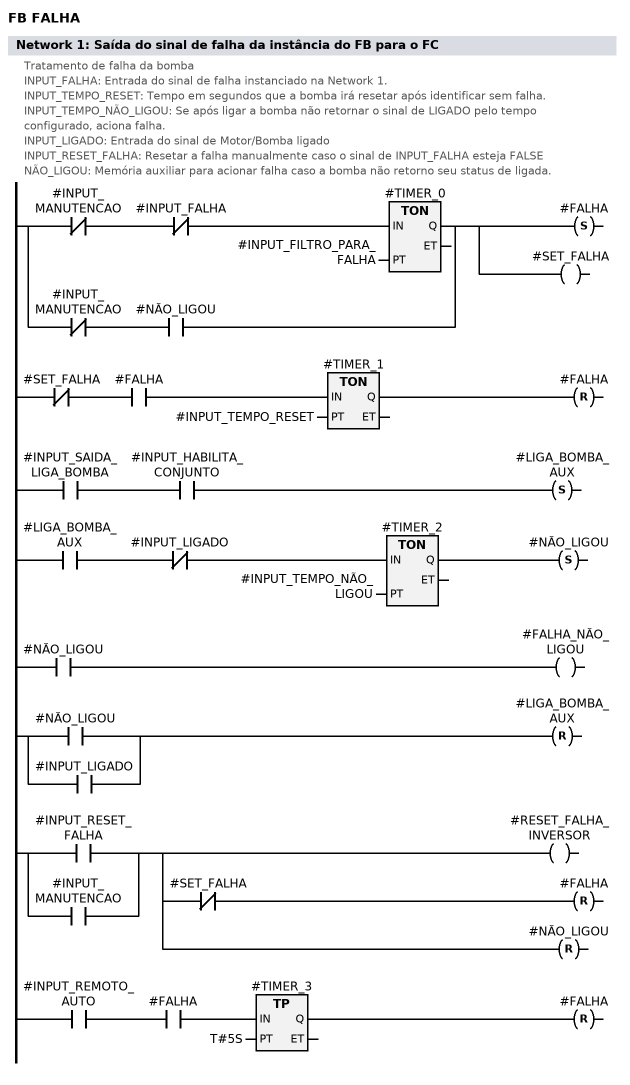
   #TIMER_0.TON(IN := NOT #INPUT_MANUTENCAO AND NOT #INPUT_FALHA, PT := #INPUT_FILTRO_PARA_FALHA);
   #_w1 := #TIMER_0.Q OR (NOT #INPUT_MANUTENCAO AND #NÃO_LIGOU);
   IF #_w1 THEN #FALHA := TRUE; END_IF;
   #SET_FALHA := #_w1;
   #TIMER_1.TON(IN := NOT #SET_FALHA AND #FALHA, PT := #INPUT_TEMPO_RESET);
   IF #TIMER_1.Q THEN #FALHA := FALSE; END_IF;
   IF #INPUT_SAIDA_LIGA_BOMBA AND #INPUT_HABILITA_CONJUNTO THEN #LIGA_BOMBA_AUX := TRUE; END_IF;
   #TIMER_2.TON(IN := #LIGA_BOMBA_AUX AND NOT #INPUT_LIGADO, PT := #INPUT_TEMPO_NÃO_LIGOU);
   IF #TIMER_2.Q THEN #NÃO_LIGOU := TRUE; END_IF;
   #FALHA_NÃO_LIGOU := #NÃO_LIGOU;
   IF #NÃO_LIGOU OR #INPUT_LIGADO THEN #LIGA_BOMBA_AUX := FALSE; END_IF;
   #RESET_FALHA_INVERSOR := #INPUT_RESET_FALHA OR #INPUT_MANUTENCAO;
   IF #RESET_FALHA_INVERSOR AND NOT #SET_FALHA THEN #FALHA := FALSE; END_IF;
   IF #RESET_FALHA_INVERSOR THEN #NÃO_LIGOU := FALSE; END_IF;
   #TIMER_3.TP(IN := #INPUT_REMOTO_AUTO AND #FALHA, PT := T#5S);
   IF #TIMER_3.Q THEN #FALHA := FALSE; END_IF;
END_REGION
END_FUNCTION_BLOCK

// folder: 1. FB Bilbiotecas/1.5 Diagnóstico

FUNCTION_BLOCK "PROFINET_DEVICE_STATES"   // FB21, SCL
{ S7_Optimized_Access := 'TRUE' }
VERSION : 0.1
   VAR_INPUT
      "Array" : Array[0..1023] of Bool;   // Array DeviceStates (1023 bools)
   END_VAR
   VAR_OUTPUT
      Word_1 : Word;   // Word 1 de saída para obter as desconecções Profinet
      Word_2 : Word;   // Word 2 de saída para obter as desconecções Profinet
   END_VAR
BEGIN
   // Word Alarmes de Desconexão Profinet

   // Word 1
   #"Word_1".%X4 := NOT #Array[4];
   #"Word_1".%X5 := NOT #Array[5];
   #"Word_1".%X6 := NOT #Array[6];
   #"Word_1".%X7 := NOT #Array[7];
   #"Word_1".%X8 := NOT #Array[8];
   #"Word_1".%X9 := NOT #Array[9];
   #"Word_1".%X10 := NOT #Array[10];
   #"Word_1".%X11 := NOT #Array[11];
   #"Word_1".%X12 := NOT #Array[12];
   #"Word_1".%X13 := NOT #Array[13];
   #"Word_1".%X14 := NOT #Array[14];
   #"Word_1".%X15 := NOT #Array[15];

   // Word 2
   #"Word_2".%X0 := NOT #Array[16];
   #"Word_2".%X1 := NOT #Array[17];
   #"Word_2".%X2 := NOT #Array[18];
   #"Word_2".%X3 := NOT #Array[19];
END_FUNCTION_BLOCK

FUNCTION_BLOCK "FB PROFINET DEVICE STATES to Word"   // FB23, SCL
{ S7_Optimized_Access := 'TRUE' }
VERSION : 0.1
   VAR_INPUT
      "Array" : Array[0..1023] of Bool;   // Array DeviceStates (1023 bools)
   END_VAR
   VAR_OUTPUT
      WORD_1 : Word;   // Word 1 de saída para obter as desconecções Profinet
      WORD_2 : Word;   // Word 2 de saída para obter as desconecções Profinet
      WORD_3 : Word;   // Word 3 de saída para obter as desconecções Profinet
      WORD_4 : Word;   // Word 4 de saída para obter as desconecções Profinet
   END_VAR
   VAR
      "word" : Array[1..4] of Word;
      i : Int;
      j : Int;
   END_VAR
BEGIN
   // Word Alarmes de Desconexão Profinet




   // Word 1
   #WORD_1.%X0 := NOT #Array[0];
   #WORD_1.%X1 := NOT #Array[1];
   #WORD_1.%X2 := NOT #Array[2];
   #WORD_1.%X3 := NOT #Array[3];
   #WORD_1.%X4 := NOT #Array[4];(*
   #WORD_1.%X5 := NOT #Array[5];
   #WORD_1.%X6 := NOT #Array[6];
   #WORD_1.%X7 := NOT #Array[7];
   #WORD_1.%X8 := NOT #Array[8];
   #WORD_1.%X9 := NOT #Array[9];*)
   #WORD_1.%X10 := NOT #Array[10];
   #WORD_1.%X11 := NOT #Array[11];
   #WORD_1.%X12 := NOT #Array[12];
   #WORD_1.%X13 := NOT #Array[13];(*
   #WORD_1.%X14 := NOT #Array[14];
   #WORD_1.%X15 := NOT #Array[15];

   //Word 2
   #WORD_2.%X0 := NOT #Array[16];
   #WORD_2.%X1 := NOT #Array[17];
   #WORD_2.%X2 := NOT #Array[18];
   #WORD_2.%X3 := NOT #Array[19];*)
   #WORD_2.%X4 := NOT #Array[20];
   #WORD_2.%X5 := NOT #Array[21];
   #WORD_2.%X6 := NOT #Array[22];
   #WORD_2.%X7 := NOT #Array[23];
   #WORD_2.%X8 := NOT #Array[24];
   #WORD_2.%X9 := NOT #Array[25];
   #WORD_2.%X10 := NOT #Array[26];
   #WORD_2.%X11 := NOT #Array[27];
   #WORD_2.%X12 := NOT #Array[28];
   #WORD_2.%X13 := NOT #Array[29];
   #WORD_2.%X14 := NOT #Array[30];
   #WORD_2.%X15 := NOT #Array[31];

   //Word 3
   #WORD_3.%X0 := NOT #Array[32];
   #WORD_3.%X1 := NOT #Array[33];
   #WORD_3.%X2 := NOT #Array[34];
   #WORD_3.%X3 := NOT #Array[35];(*
   #WORD_3.%X4 := NOT #Array[36];
   #WORD_3.%X5 := NOT #Array[37];
   #WORD_3.%X6 := NOT #Array[38];
   #WORD_3.%X7 := NOT #Array[39];*)
   #WORD_3.%X8 := NOT #Array[40];
   #WORD_3.%X9 := NOT #Array[41];
   #WORD_3.%X10 := NOT #Array[42];
   #WORD_3.%X11 := NOT #Array[43];
   #WORD_3.%X12 := NOT #Array[44];
   #WORD_3.%X13 := NOT #Array[45];
   #WORD_3.%X14 := NOT #Array[46];
   #WORD_3.%X15 := NOT #Array[47];

   //Word 4
   #WORD_4.%X0 := NOT #Array[48];(*
   #WORD_4.%X1 := NOT #Array[49];*)
   #WORD_4.%X2 := NOT #Array[50];
   #WORD_4.%X3 := NOT #Array[51];
   #WORD_4.%X4 := NOT #Array[52];
   #WORD_4.%X5 := NOT #Array[53];
   #WORD_4.%X6 := NOT #Array[54];
   #WORD_4.%X7 := NOT #Array[55];
   #WORD_4.%X8 := NOT #Array[56];
   #WORD_4.%X9 := NOT #Array[57];
   #WORD_4.%X10 := NOT #Array[58];
   #WORD_4.%X11 := NOT #Array[59];
   #WORD_4.%X12 := NOT #Array[60];
   #WORD_4.%X13 := NOT #Array[61];(*
   #WORD_4.%X14 := NOT #Array[62];
   #WORD_4.%X15 := NOT #Array[63];*)
END_FUNCTION_BLOCK

FUNCTION_BLOCK "FB PROFINET DEVICE STATES to BIT"   // FB26, SCL
{ S7_Optimized_Access := 'TRUE' }
VERSION : 0.1
   VAR_INPUT
      "Array" : Array[0..1023] of Bool;   // Array DeviceStates (1023 bools)
   END_VAR
   VAR_OUTPUT
      Bit_1 : Bool;   // Word 1 de saída para obter as desconecções Profinet
      Bit_2 : Bool;   // Word 2 de saída para obter as desconecções Profinet
      Bit_3 : Bool;   // Word 3 de saída para obter as desconecções Profinet
      Bit_4 : Bool;   // Word 4 de saída para obter as desconecções Profinet
      Bit_5 : Bool;
      Bit_6 : Bool;
      Bit_7 : Bool;
      Bit_8 : Bool;
      Bit_9 : Bool;
      Bit_10 : Bool;
      Bit_11 : Bool;
      Bit_12 : Bool;
      Bit_13 : Bool;
      Bit_14 : Bool;
      Bit_15 : Bool;
      Bit_16 : Bool;
      Bit_17 : Bool;
      Bit_18 : Bool;
      Bit_19 : Bool;
      Bit_20 : Bool;
      Bit_21 : Bool;
      Bit_22 : Bool;
      Bit_23 : Bool;
      Bit_24 : Bool;
      Bit_25 : Bool;
      Bit_26 : Bool;
      Bit_27 : Bool;
      Bit_28 : Bool;
      Bit_29 : Bool;
      Bit_30 : Bool;
      Bit_31 : Bool;
      Bit_32 : Bool;
      Bit_33 : Bool;
      Bit_34 : Bool;
      Bit_35 : Bool;
      Bit_36 : Bool;
      Bit_37 : Bool;
      Bit_38 : Bool;
      Bit_39 : Bool;
      Bit_40 : Bool;
      Bit_41 : Bool;
      Bit_42 : Bool;
      Bit_43 : Bool;
      Bit_44 : Bool;
      Bit_45 : Bool;
      Bit_46 : Bool;
      Bit_47 : Bool;
      Bit_48 : Bool;
      Bit_49 : Bool;
      Bit_50 : Bool;
      Bit_51 : Bool;
      Bit_52 : Bool;
      Bit_53 : Bool;
      Bit_54 : Bool;
      Bit_55 : Bool;
      Bit_56 : Bool;
      Bit_57 : Bool;
      Bit_58 : Bool;
      Bit_59 : Bool;
      Bit_60 : Bool;
      Bit_61 : Bool;
      Bit_62 : Bool;
      Bit_63 : Bool;
      Bit_64 : Bool;
   END_VAR
   VAR
      "word" : Array[1..4] of Word;
      i : Int;
      j : Int;
   END_VAR
BEGIN
   #Bit_1 :=  #Array[0];
   #Bit_2 :=  #Array[1];
   #Bit_3 :=  #Array[2];
   #Bit_4 :=  #Array[3];
   #Bit_5 :=  #Array[4];
   #Bit_6 :=  #Array[5];
   #Bit_7 :=  #Array[6];
   #Bit_8 :=  #Array[7];
   #Bit_9 :=  #Array[8];
   #Bit_10 :=  #Array[9];
   #Bit_11 :=  #Array[10];
   #Bit_12 :=  #Array[11];
   #Bit_13 :=  #Array[12];
   #Bit_14 :=  #Array[13];
   #Bit_15 :=  #Array[14];
   #Bit_16 :=  #Array[15];
   #Bit_17 :=  #Array[16];
   #Bit_18 :=  #Array[17];
   #Bit_19 :=  #Array[18];
   #Bit_20 :=  #Array[19];
   #Bit_21 :=  #Array[20];
   #Bit_22 :=  #Array[21];
   #Bit_23 :=  #Array[22];
   #Bit_24 :=  #Array[23];
   #Bit_25 :=  #Array[24];
   #Bit_26 :=  #Array[25];
   #Bit_27 :=  #Array[26];
   #Bit_28 :=  #Array[27];
   #Bit_29 :=  #Array[28];
   #Bit_30 :=  #Array[29];
   #Bit_31 :=  #Array[30];
   #Bit_32 :=  #Array[31];
   #Bit_33 :=  #Array[32];
   #Bit_34 :=  #Array[33];
   #Bit_35 :=  #Array[34];
   #Bit_36 :=  #Array[35];
   #Bit_37 :=  #Array[36];
   #Bit_38 :=  #Array[37];
   #Bit_39 :=  #Array[38];
   #Bit_40 :=  #Array[39];
   #Bit_41 :=  #Array[40];
   #Bit_42 :=  #Array[41];
   #Bit_43 :=  #Array[42];
   #Bit_44 :=  #Array[43];
   #Bit_45 :=  #Array[44];
   #Bit_46 :=  #Array[45];
   #Bit_47 :=  #Array[46];
   #Bit_48 :=  #Array[47];
   #Bit_49 :=  #Array[48];
   #Bit_50 :=  #Array[49];
   #Bit_51 :=  #Array[50];
   #Bit_52 :=  #Array[51];
   #Bit_53 :=  #Array[52];
   #Bit_54 :=  #Array[53];
   #Bit_55 :=  #Array[54];
   #Bit_56 :=  #Array[55];
   #Bit_57 :=  #Array[56];
   #Bit_58 :=  #Array[57];
   #Bit_59 :=  #Array[58];
   #Bit_60 :=  #Array[59];
   #Bit_61 :=  #Array[60];
   #Bit_62 :=  #Array[61];
   #Bit_63 :=  #Array[62];
   #Bit_64 :=  #Array[63];
END_FUNCTION_BLOCK

FUNCTION_BLOCK "FB DIAG MODULES"   // FB28, LAD
{ S7_Optimized_Access := 'TRUE' }
VERSION : 0.1
   VAR_INPUT
      LADDR : HW_ANY;   // ID de hardware do componente de hardware
      MODE : UInt;   // Use o parâmetro de modo para selecionar quais dados de diagnóstico são emitidos.
   END_VAR
   VAR_OUTPUT
      "OUT_WORD[bit]" : Bool;   // Bit da Word de saída representando falha/avaria do dispositivo
      Maintence_State : String;
      Component_StateDetail : String;
      Own_State : String;
      IO_State : String;
      Operating_State : String;
      Ret_Val : String;
   END_VAR
   VAR
      "Maintence State" : Array[0..10] of String;
      ComponentStateDetail : Array[0..31] of String;
      OwnState : Array[0..7] of String;
      IOState : Array[0..15] of String;
      OperatingState : Array[0..40] of String;
      DIAG : DIS;
      CNT_DIAG : UInt;
      RET_VAL_STRING : Array[0..6] of String;
      RET_VAL_1 : Int;
   END_VAR
   // "Maintence State"[0] := 'Good';
   // "Maintence State"[1] := 'The hardware component is disabled.';
   // "Maintence State"[5] := 'Maintenance required';
   // "Maintence State"[6] := 'Maintenance demanded';
   // "Maintence State"[7] := 'Error';
   // "Maintence State"[8] := 'Status unknown / error in higher-level hardware component';
   // "Maintence State"[10] := 'Inputs/outputs are not available.';
   // ComponentStateDetail[3] := 'least one qualified diagnostics is available';
   // ComponentStateDetail[4] := 'Maintenance required for at least one channel or the component';
   // ComponentStateDetail[5] := 'Maintenance demanded for at least one channel or the component';
   // ComponentStateDetail[6] := 'Error in at least one channel or the component';
   // ComponentStateDetail[7] := 'Application Ready Pending - No I/O access';
   // ComponentStateDetail[8] := 'Locked by Superordinated - No access to hardware component';
   // ComponentStateDetail[9] := 'Locked by IOController - No access to hardware component';
   // ComponentStateDetail[10] := 'Locked by IOSupervisor - No access to hardware component';
   // ComponentStateDetail[16] := 'Submodule or module disabled';
   // ComponentStateDetail[17] := 'CiR operation active';
   // ComponentStateDetail[18] := 'Input not available';
   // ComponentStateDetail[19] := 'Output not available';
   // ComponentStateDetail[20] := 'Overflow diagnostics buffer';
   // ComponentStateDetail[21] := 'Diagnostics not available';
   // ComponentStateDetail[22] := 'Partial device failure (with PNIO for Shared iDevices)';
   // OwnState[0] := 'Good';
   // OwnState[1] := 'Disabled';
   // OwnState[2] := 'Maintenance required';
   // OwnState[3] := 'Maintenance demanded';
   // OwnState[4] := 'Error';
   // OwnState[5] := 'Not accessible';
   // OwnState[6] := 'Diagnostic status unknown';
   // OwnState[7] := 'IO not available - Inputs/outputs are not available.';
   // IOState[0] := 'Good';
   // IOState[1] := 'Disabled';
   // IOState[2] := 'Maintenance required';
   // IOState[3] := 'Maintenance demanded';
   // IOState[4] := 'Error';
   // IOState[5] := 'Hardware component not reachable - Hardware component cannot be accessed.';
   // IOState[6] := 'Qualified: Bit 6 = 1 if at least one qualified diagnostics is available';
   // IOState[7] := 'I/O data not available - I/O data not available';
   // IOState[14] := 'Network error';
   // IOState[15] := 'Hardware error';
   // OperatingState[1] := 'STOP / firmware update';
   // OperatingState[2] := 'STOP / Memory reset';
   // OperatingState[3] := 'STOP / self start';
   // OperatingState[4] := 'STOP';
   // OperatingState[5] := 'Memory reset';
   // OperatingState[6] := 'Startup';
   // OperatingState[8] := 'RUN';
   // OperatingState[9] := 'RUN-Redundant';
   // OperatingState[10] := 'HOLD';
   // OperatingState[13] := 'DEFECT (Note: can only be seen in diagnostics buffer entries)';
   // OperatingState[15] := 'De-energized (Note: can only be seen in diagnostics buffer entries)';
   // OperatingState[16] := 'CiR';
   // OperatingState[17] := 'STOP without ODIS';
   // OperatingState[18] := 'RUN ODIS';
   // OperatingState[19] := 'PgmTest';
   // OperatingState[20] := 'RunPgmTest (state of primary CPU when the backup CPU is in test mode)';
   // OperatingState[21] := 'Run-Syncup (only Primary CPU in SYNCUP system state)';
   // OperatingState[22] := 'SYNCUP (only backup CPU in SYNCUP system state)';
   // OperatingState[31] := 'State of partner CPU unknown (for example when the partner CPU is not available)';
   // OperatingState[33] := 'STOP system state';
   // OperatingState[35] := 'STARTUP system state';
   // OperatingState[37] := 'RUN-Solo system state';
   // OperatingState[38] := 'SYNCUP system state';
   // OperatingState[40] := 'RUN-Redundant system state';
   // RET_VAL_STRING[0] := 'Feedback signal ok';
   // RET_VAL_STRING[1] := 'The data area at the DETAIL parameter is too small. Not all details of the diagnostics data are output.';
   // RET_VAL_STRING[2] := 'Value in the MODE parameter is not supported.';
   // RET_VAL_STRING[3] := 'Type at the DIAG parameter is not supported with the selected mode (parameter MODE).';
   // RET_VAL_STRING[4] := 'Type at the DETAIL parameter is not supported with the selected mode (parameter MODE).';
   // RET_VAL_STRING[5] := 'LADDR does not exist';
   // RET_VAL_STRING[6] := 'Insufficient resources for parallel execution.';
BEGIN

REGION Network 1
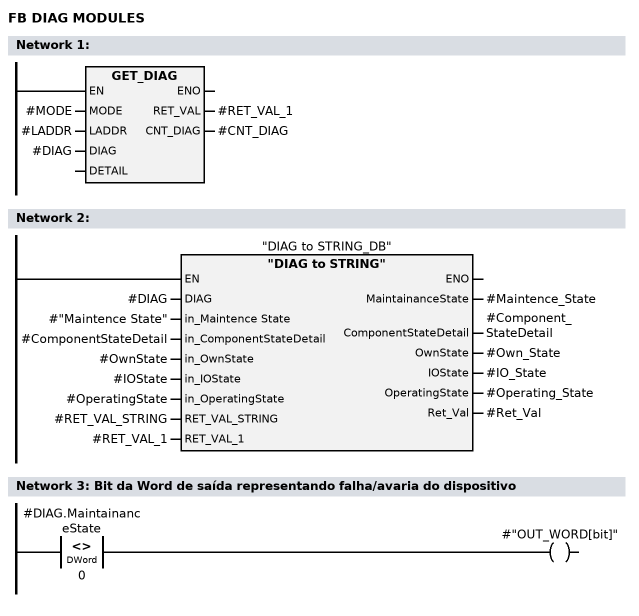
   #RET_VAL_1 := GET_DIAG(MODE := #MODE, LADDR := #LADDR, DIAG := #DIAG, CNT_DIAG => #CNT_DIAG);
END_REGION

REGION Network 2
   RUNG wire#powerrail
      "DIAG to STRING_DB"(DIAG := #DIAG, "in_Maintence State" := #"Maintence State", in_ComponentStateDetail := #ComponentStateDetail, in_OwnState := #OwnState, in_IOState := #IOState, in_OperatingState := #OperatingState, RET_VAL_STRING := #RET_VAL_STRING, RET_VAL_1 := #RET_VAL_1, MaintainanceState => #Maintence_State, ComponentStateDetail => #Component_StateDetail, OwnState => #Own_State, IOState => #IO_State, OperatingState => #Operating_State, Ret_Val => #Ret_Val)
   END_RUNG
   // the same network as SCL:
   "DIAG to STRING_DB"(DIAG := #DIAG,   // "DIAG to STRING"
                       "in_Maintence State" := #"Maintence State",
                       in_ComponentStateDetail := #ComponentStateDetail,
                       in_OwnState := #OwnState,
                       in_IOState := #IOState,
                       in_OperatingState := #OperatingState,
                       RET_VAL_STRING := #RET_VAL_STRING,
                       RET_VAL_1 := #RET_VAL_1,
                       MaintainanceState => #Maintence_State,
                       ComponentStateDetail => #Component_StateDetail,
                       OwnState => #Own_State,
                       IOState => #IO_State,
                       OperatingState => #Operating_State,
                       Ret_Val => #Ret_Val);
END_REGION

REGION Network 3: Bit da Word de saída representando falha/avaria do dispositivo
   RUNG wire#powerrail
      { S7_Templates := "SrcType := DWord" } NE_Contact(in1 := #DIAG.MaintainanceState, in2 := 0)
      Coil( #"OUT_WORD[bit]" )
   END_RUNG
   // the same network as SCL:
   #"OUT_WORD[bit]" := #DIAG.MaintainanceState <> 0;
END_REGION
END_FUNCTION_BLOCK

FUNCTION_BLOCK "DIAG to STRING"   // FB29, SCL
{ S7_Optimized_Access := 'TRUE' }
VERSION : 0.1
   VAR_INPUT
      DIAG : DIS;
      "in_Maintence State" : Array[0..10] of String;
      in_ComponentStateDetail : Array[0..31] of String;
      in_OwnState : Array[0..7] of String;
      in_IOState : Array[0..15] of String;
      in_OperatingState : Array[0..40] of String;
      RET_VAL_STRING : Array[0..6] of String;
      RET_VAL_1 : UInt;
   END_VAR
   VAR_OUTPUT
      MaintainanceState : String[254];
      ComponentStateDetail : String[254];
      OwnState : String[254];
      IOState : String[254];
      OperatingState : String[254];
      Ret_Val : String[254];
   END_VAR
   VAR
      i : Int;
      j : UInt;
      k : UInt;
      "m" : UInt;
      n : UInt;
      o : UInt;
      Separator : String[5];
   END_VAR
BEGIN
   // PARA MaintainanceState
   FOR #i := 0 TO 10 DO
       IF #DIAG.MaintainanceState = #i THEN
           #MaintainanceState := #"in_Maintence State"[#i];
       END_IF;
   END_FOR;

   #Separator := '; ';
   #ComponentStateDetail := '';
   #IOState := '';
   FOR #j := 0 TO 31 DO
       // testa se o bit #j está 1
       IF (#DIAG.ComponentStateDetail AND SHL(IN:= DWORD#1, N:= #j)) <> DWORD#0 THEN
           // ignora entradas vazias
           IF LEN(#in_ComponentStateDetail[#j]) > 0 THEN
               // separador só se já houver conteúdo
               IF LEN(#ComponentStateDetail) > 0 THEN
                   #ComponentStateDetail := CONCAT(IN1 := #ComponentStateDetail, IN2 := #Separator);
               END_IF;
               // concatena o texto do índice ativo
               #ComponentStateDetail := CONCAT(IN1 := #ComponentStateDetail, IN2 := #in_ComponentStateDetail[#j]);
           END_IF;
       END_IF;
   END_FOR;

   FOR #k := 0 TO 7 DO
       IF #DIAG.OwnState = #k THEN
           #OwnState := #in_OwnState[#k];
       END_IF;
   END_FOR;

   FOR #m := 0 TO 15 DO
       IF (#DIAG.IOState AND SHL(IN := DWORD#1, N := #m)) <> DWORD#0 THEN
           IF LEN(#in_IOState[#m]) > 0 THEN
               IF LEN(#IOState) > 0 THEN
                   #IOState := CONCAT(IN1 := #IOState, IN2 := #Separator);
               END_IF;
               #IOState := CONCAT(IN1 := #IOState, IN2 := #in_IOState[#m]);
           END_IF;
       END_IF;
   END_FOR;

   FOR #n := 0 TO 40 DO
       IF #DIAG.OperatingState = #n THEN
           #OperatingState := #in_OperatingState[#i];
       END_IF;
   END_FOR;

   CASE #RET_VAL_1 OF
       UINT#16#0000:
           #Ret_Val := #RET_VAL_STRING[0];
       UINT#16#8080:
           #Ret_Val := #RET_VAL_STRING[2];
       UINT#16#8081:
           #Ret_Val := #RET_VAL_STRING[3];
       UINT#16#8082:
           #Ret_Val := #RET_VAL_STRING[4];
       UINT#16#8090:
           #Ret_Val := #RET_VAL_STRING[5];
       UINT#16#80C1:
           #Ret_Val := #RET_VAL_STRING[6];

       ELSE
           #Ret_Val := #RET_VAL_STRING[2];  // default
   END_CASE;
END_FUNCTION_BLOCK

// folder: 1. FB Bilbiotecas/1.6 Comunicação Modbus

FUNCTION_BLOCK "FB MODBUS MASTER BLOCK MMW"   // FB18, LAD
{ S7_Optimized_Access := 'TRUE' }
VERSION : 0.1
// Instanciamento do Bloco Modbus Master para cada Driver (Multimedidor)
// 
// Network 1: Chamada por índice de endereço
// Network 2: Falha de comunicação Modbus
// Network 3: Reset do módulo de comunicação Modbus
   VAR_INPUT
      INDEX_DRIVER : Int;   // Índice do driver, numerando a instância de cada um
      INDEX_ADDR : Int;   // Índice do endereço, numerando a ordem de leitura de cada um
      TRIGGER : Bool;   // Gatilho de chamada do bloco. (Recebido da instância do FB SCAN DRIVERS conforme o DONE do bloco master)
      MODBUS_ID : Int;   // Endereço ID do Modbus
      ARRAY_ADDR_MMW : Array[0..38] of Int;   // Array de endereços (Todos os 41 endereços cadastrados na tabela Modbus do equipamento)
      INDEX_BLOCK : Int;   // Índice de instância, para definir quando os blocos Master serão chamados
      CICLE_TIMES_SET_ALARME : Int;   // Cadastro do "Tryout", número de tentativas de comunicação antes de acionar o erro
   END_VAR
   VAR_OUTPUT
      DRIVER_ERROR_COMUNIC : Bool;   // Erro de comunicação Modbus
      ERROR_CODE : Word;   // Código do erro de comunicação Modbus
      RESET_PTP : Bool;   // Saída para reset do módulo Commload
   END_VAR
   VAR_IN_OUT
      MODBUS_MASTER : Modbus_Master;
      ARRAY_MMW : Array[0..38] of Real;   // Array da DB GLOBAL onde os registros são armazenados
   END_VAR
   VAR
      PULSE_SCAN : Bool;   // Pulso para contagem do número de tentativas de comunicação mal sucedidas
      COUT_PULSE : Bool;   // Memória auxiliar do pulso
      ERROR_CICLES : Int;   // Memória de incremento a cada pulso do PULSE_SCAN
      ACTUAL_ERROR : Word;   // Captura do código de erro na tentativa de comunicação mal sucedida
      MASTER_DRIVER_LAST_ERROR : Int;   // Índice do driver que registrou o último erro
      ARRAY_READ_MMW : Array[0..254] of Real;   // Array local para armazenar temporariamente as leituras antes de mover à DB GLOBAL
      HABILITA_RESET : Bool;   // Habilita reset após intervalo de tempo
      AUX_RESET : Bool;   // Memória auxiliar para o reset modbus
      RESET_TIMER_1 : IEC_TIMER;   // Tempo de cooldown para utilizar o reset novamente
      RESET_TIMER_2 : IEC_TIMER;   // Tempo de saída acionada (reset)
   END_VAR
   VAR_TEMP   // added for the SCL form of the ladder/FBD networks
      _w1 : Bool;
      _w2 : Bool;
   END_VAR
BEGIN

REGION Network 1: Function BLock MODBUS MASTER BLOCK MMW
   // Ao chamar o bloco, o índice de endereço irá alternar entre os 41 endereços do multimedidor. Essas informações são registradas em um array de tamanho 41 e movidos à DB GLOBAL.
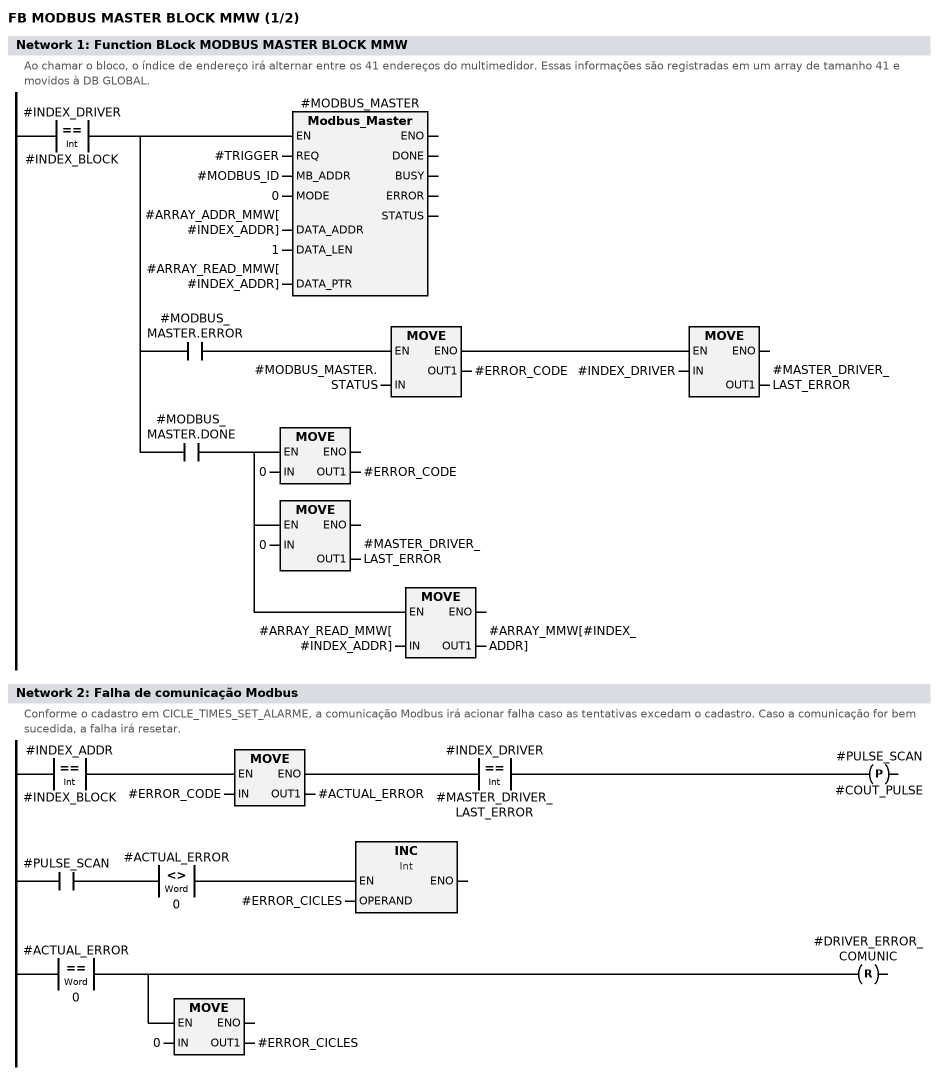
   #_w1 := #INDEX_DRIVER = #INDEX_BLOCK;
   IF #_w1 THEN
       #MODBUS_MASTER(REQ := #TRIGGER,   // Modbus_Master
                      MB_ADDR := #MODBUS_ID,
                      MODE := 0,
                      DATA_ADDR := #ARRAY_ADDR_MMW[#INDEX_ADDR],
                      DATA_LEN := 1,
                      DATA_PTR := #ARRAY_READ_MMW[#INDEX_ADDR]);
   END_IF;
   IF #_w1 AND #MODBUS_MASTER.ERROR THEN
       #ERROR_CODE := #MODBUS_MASTER.STATUS;
       #MASTER_DRIVER_LAST_ERROR := #INDEX_DRIVER;
   END_IF;
   IF #_w1 AND #MODBUS_MASTER.DONE THEN
       #ERROR_CODE := 0;
       #MASTER_DRIVER_LAST_ERROR := 0;
       #ARRAY_MMW[#INDEX_ADDR] := #ARRAY_READ_MMW[#INDEX_ADDR];
   END_IF;
END_REGION

REGION Network 2: Falha de comunicação Modbus
   // Conforme o cadastro em CICLE_TIMES_SET_ALARME, a comunicação Modbus irá acionar falha caso as tentativas excedam o cadastro. Caso a comunicação for bem sucedida, a falha irá resetar.
   #_w1 := #INDEX_ADDR = #INDEX_BLOCK;
   IF #_w1 THEN #ACTUAL_ERROR := #ERROR_CODE; END_IF;
   #_w2 := #_w1 AND (#INDEX_DRIVER = #MASTER_DRIVER_LAST_ERROR);
   #PULSE_SCAN := #_w2 AND NOT #COUT_PULSE;   // rising edge
   #COUT_PULSE := #_w2;
   IF #PULSE_SCAN AND (#ACTUAL_ERROR <> 0) THEN #ERROR_CICLES := #ERROR_CICLES + 1; END_IF;
   IF #ACTUAL_ERROR = 0 THEN
       #DRIVER_ERROR_COMUNIC := FALSE;
       #ERROR_CICLES := 0;
   END_IF;
END_REGION

REGION Network 3: Reset do módulo de comunicação Modbus
   // Reset ao identificar erro de comunicação.
   // Tempo de cooldown 600s (10min): Intervalo de tempo após o reset para resetar novamente caso o equipamento ainda esteja em erro.
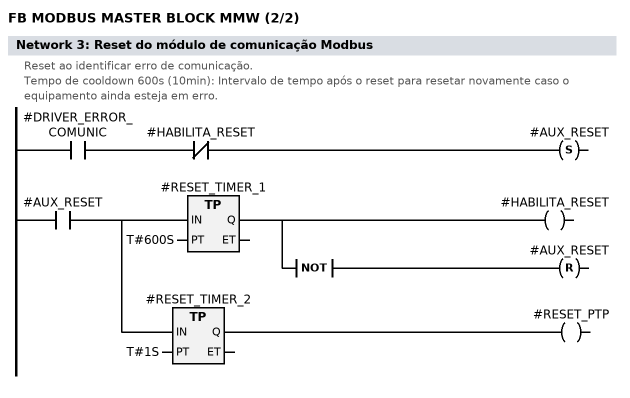
   IF #DRIVER_ERROR_COMUNIC AND NOT #HABILITA_RESET THEN #AUX_RESET := TRUE; END_IF;
   #RESET_TIMER_1.TP(IN := #AUX_RESET, PT := T#600S);
   #HABILITA_RESET := #RESET_TIMER_1.Q;
   #_w1 := #AUX_RESET;
   IF NOT #RESET_TIMER_1.Q THEN #AUX_RESET := FALSE; END_IF;
   #RESET_TIMER_2.TP(IN := #_w1, PT := T#1S);
   #RESET_PTP := #RESET_TIMER_2.Q;
END_REGION
END_FUNCTION_BLOCK

FUNCTION_BLOCK "FB MODBUS MASTER BLOCK"   // FB19, LAD
TITLE = Function Block MODBUS MASTER BLOCK
{ S7_Optimized_Access := 'TRUE' }
VERSION : 0.1
// Instanciamento do Bloco Modbus Master para cada Driver (Inversor ou rádio)
// 
// Network 1: Chamada por índice de endereço
// Network 2: Falha de comunicação Modbus
// Network 3: Segundeiro, segundos sem comunicação
// Network 4: Reset do módulo de comunicação Modbus
   VAR_INPUT
      INDEX_DRIVER : Int;   // Índice do driver, numerando a instância de cada um
      INDEX_ADDR : Int;   // Índice do endereço, numerando a ordem de leitura de cada um
      TRIGGER : Bool;   // Gatilho de chamada do bloco. (Recebido da instância do FB SCAN DRIVERS conforme o DONE do bloco master)
      MODBUS_ID : Int;   // Endereço ID do Modbus
      DATA_ADDR_1 : DInt;   // Endereço 1 para acesso à tabela modbus
      MODE_ADDR_1 : Byte;   // Modo (0 = Leitura, 1 = Escrita)
      DATA_LEN_1 : Byte;
      IS_MMW_2 : Bool;
      DATA_ADDR_2 : DInt;   // Endereço 2 para acesso à tabela modbus
      MODE_ADDR_2 : Byte;   // Modo (0 = Leitura, 1 = Escrita)
      DATA_LEN_2 : Byte;
      IS_MMW_3 : Bool;
      DATA_ADDR_3 : DInt;   // Endereço 3 para acesso à tabela modbus
      MODE_ADDR_3 : Byte;   // Modo (0 = Leitura, 1 = Escrita)
      DATA_LEN_3 : Byte;
      IS_MMW_4 : Bool;
      DATA_ADDR_4 : DInt;   // Endereço 3 para acesso à tabela modbus
      MODE_ADDR_4 : Byte;   // Modo (0 = Leitura, 1 = Escrita)
      DATA_LEN_4 : Byte;
      IS_MMW_5 : Bool;
      DATA_ADDR_5 : DInt;   // Endereço 3 para acesso à tabela modbus
      MODE_ADDR_5 : Byte;   // Modo (0 = Leitura, 1 = Escrita)
      DATA_LEN_5 : Byte;
      INDEX_BLOCK : Int;   // Índice de instância, para definir quando os blocos Master serão chamados
      CICLE_TIMES_SET_ALARME : Int;   // Cadastro do "Tryout", número de tentativas de comunicação antes de acionar o erro
   END_VAR
   VAR_OUTPUT
      DRIVER_ERROR_COMUNIC : Bool;   // Erro de comunicação Modbus
      ERROR_CODE : Word;   // Código do erro de comunicação Modbus
      ERROR_CICLES : Int;   // Memória de incremento a cada pulso do PULSE_SCAN
      SEGUNDEIRO : Int;   // Segundos sem comunicação
      RESET_PTP : Bool;   // Saída para reset do módulo Commload
   END_VAR
   VAR_IN_OUT
      MODBUS_MASTER : Modbus_Master;   // Entrada do Bloco Master na instância
      DATA_PTR_1 : Variant;   // Endereço da DB GLOBAL onde a leitura proveninente do DATA_ADDR_1 é armazenada
      DATA_PTR_2 : Variant;   // Endereço da DB GLOBAL onde a leitura proveninente do DATA_ADDR_2 é armazenada
      DATA_PTR_3 : Variant;   // Endereço da DB GLOBAL onde a leitura proveninente do DATA_ADDR_3 é armazenada
      DATA_PTR_4 : Variant;   // Endereço da DB GLOBAL onde a leitura proveninente do DATA_ADDR_3 é armazenada
      DATA_PTR_5 : Variant;   // Endereço da DB GLOBAL onde a leitura proveninente do DATA_ADDR_3 é armazenada
   END_VAR
   VAR
      PULSE_SCAN : Bool;   // Pulso para contagem do número de tentativas de comunicação mal sucedidas
      COUNT_PULSE : Bool;   // Memória auxiliar do pulso
      ACTUAL_ERROR : Word;   // Captura do código de erro na tentativa de comunicação mal sucedida
      MASTER_DRIVER_LAST_ERROR : Int;   // Índice do driver que registrou o último erro
      ERROR_MASTER_1 : Bool;   // Código de erro do mestre 1 (addr 1)
      ERROR_MASTER_2 : Bool;   // Código de erro do mestre 2 (addr 2)
      ERROR_MASTER_3 : Bool;   // Código de erro do mestre 3 (addr 3)
      ERROR_MASTER_4 : Bool;   // Código de erro do mestre 3 (addr 3)
      ERROR_MASTER_5 : Bool;   // Código de erro do mestre 3 (addr 3)
      STATUS_MASTER_1 : Word;   // Status do mestre 1 (addr 1)
      STATUS_MASTER_2 : Word;   // Status do mestre 2 (addr 2)
      STATUS_MASTER_3 : Word;   // Status do mestre 3 (addr 3)
      STATUS_MASTER_4 : Word;   // Status do mestre 3 (addr 3)
      STATUS_MASTER_5 : Word;   // Status do mestre 3 (addr 3)
      DONE : Bool;   // Indicador de comunicação bem sucedida
      DONE_PULSO : Int;   // Pulso de comunicação bem sucedida
      SEGUNDEIRO_PULSO : Bool;   // Pulso para contar os segundos sem comunicação
      SEGUNDEIRO_AUX : Bool;   // Memória auxiliar do segundeiro
      HABILITA_RESET : Bool;   // Habilita reset após intervalo de tempo
      AUX_RESET : Bool;   // Memória auxiliar para o reset modbus
      SET_COOLDOWN : Bool;   // Memória Auxiliar do Cooldown Timer
      RESET_COOLDOWN : Bool;   // Memória Auxiliar do Cooldown Timer
      RESET_TIMER_1 : IEC_TIMER;   // Tempo de cooldown para utilizar o reset novamente
      RESET_TIMER_2 : IEC_TIMER;   // Tempo de saída acionada (reset)
      COOLDOWN_TIMER_1 : IEC_TIMER;   // Tempo para resetar os ciclos sem comunicação
      COOLDOWN_TIMER_2 : IEC_TIMER;   // Tempo de espera após reset para resetar novamente
      COOLDOWN_TIMER_3 : IEC_TIMER;
   END_VAR
   VAR_TEMP   // added for the SCL form of the ladder/FBD networks
      _w1 : Bool;
      _w2 : Bool;
   END_VAR
BEGIN

REGION Network 1: Chamada por índice de endereço
   // Cada vez que o bloco Master é chamado, um índice de endereço diferente é armazenado.
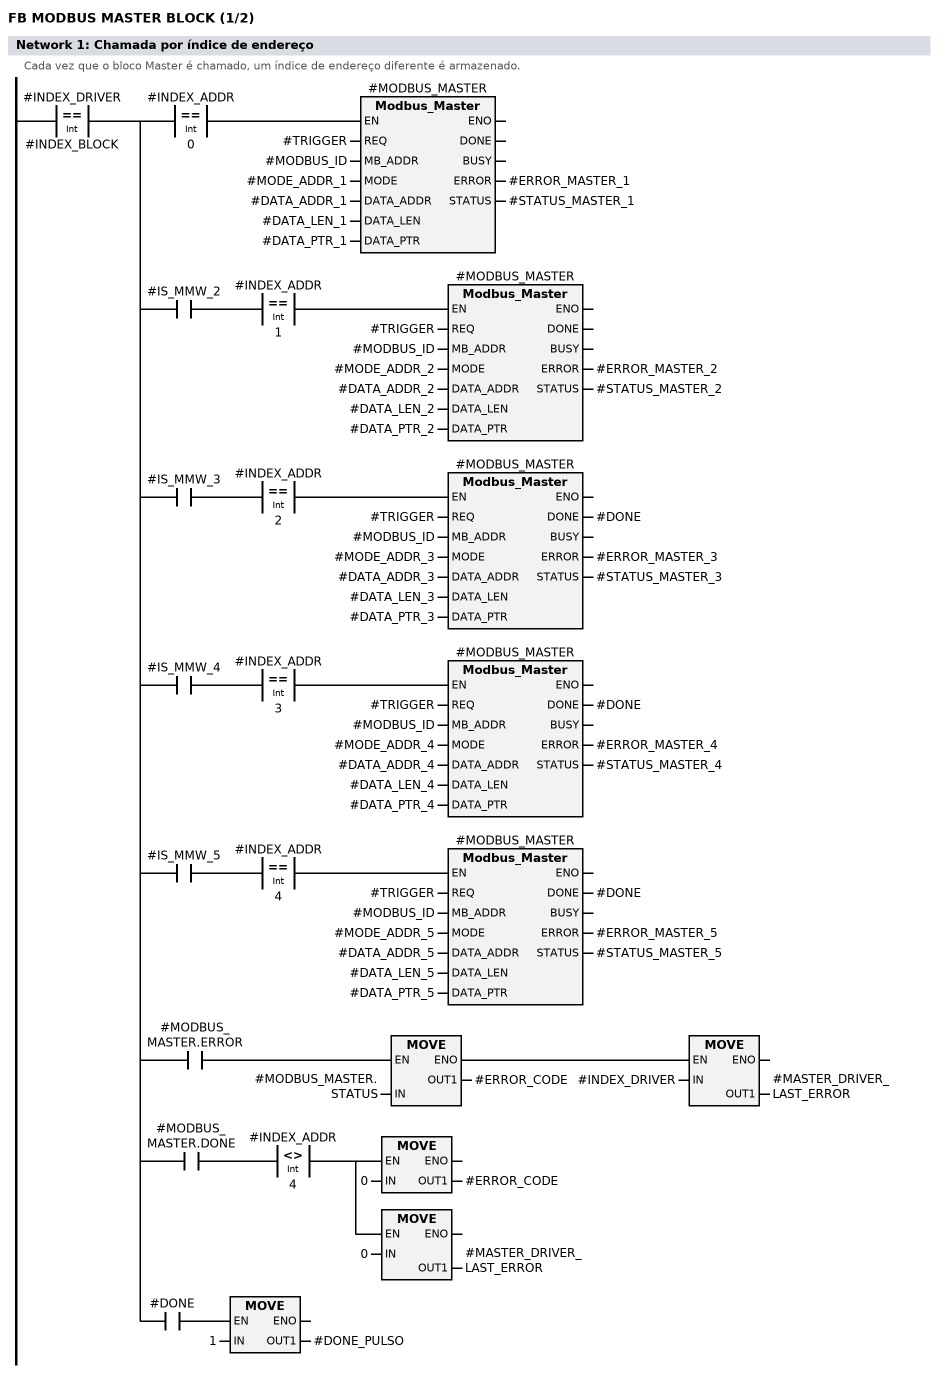
   #_w1 := #INDEX_DRIVER = #INDEX_BLOCK;
   IF #_w1 AND (#INDEX_ADDR = 0) THEN
       #MODBUS_MASTER(REQ := #TRIGGER,   // Modbus_Master
                      MB_ADDR := #MODBUS_ID,
                      MODE := #MODE_ADDR_1,
                      DATA_ADDR := #DATA_ADDR_1,
                      DATA_LEN := #DATA_LEN_1,
                      DATA_PTR := #DATA_PTR_1,
                      ERROR => #ERROR_MASTER_1,
                      STATUS => #STATUS_MASTER_1);
   END_IF;
   IF #_w1 AND #IS_MMW_2 AND (#INDEX_ADDR = 1) THEN
       #MODBUS_MASTER(REQ := #TRIGGER,   // Modbus_Master
                      MB_ADDR := #MODBUS_ID,
                      MODE := #MODE_ADDR_2,
                      DATA_ADDR := #DATA_ADDR_2,
                      DATA_LEN := #DATA_LEN_2,
                      DATA_PTR := #DATA_PTR_2,
                      ERROR => #ERROR_MASTER_2,
                      STATUS => #STATUS_MASTER_2);
   END_IF;
   IF #_w1 AND #IS_MMW_3 AND (#INDEX_ADDR = 2) THEN
       #MODBUS_MASTER(REQ := #TRIGGER,   // Modbus_Master
                      MB_ADDR := #MODBUS_ID,
                      MODE := #MODE_ADDR_3,
                      DATA_ADDR := #DATA_ADDR_3,
                      DATA_LEN := #DATA_LEN_3,
                      DATA_PTR := #DATA_PTR_3,
                      DONE => #DONE,
                      ERROR => #ERROR_MASTER_3,
                      STATUS => #STATUS_MASTER_3);
   END_IF;
   IF #_w1 AND #IS_MMW_4 AND (#INDEX_ADDR = 3) THEN
       #MODBUS_MASTER(REQ := #TRIGGER,   // Modbus_Master
                      MB_ADDR := #MODBUS_ID,
                      MODE := #MODE_ADDR_4,
                      DATA_ADDR := #DATA_ADDR_4,
                      DATA_LEN := #DATA_LEN_4,
                      DATA_PTR := #DATA_PTR_4,
                      DONE => #DONE,
                      ERROR => #ERROR_MASTER_4,
                      STATUS => #STATUS_MASTER_4);
   END_IF;
   IF #_w1 AND #IS_MMW_5 AND (#INDEX_ADDR = 4) THEN
       #MODBUS_MASTER(REQ := #TRIGGER,   // Modbus_Master
                      MB_ADDR := #MODBUS_ID,
                      MODE := #MODE_ADDR_5,
                      DATA_ADDR := #DATA_ADDR_5,
                      DATA_LEN := #DATA_LEN_5,
                      DATA_PTR := #DATA_PTR_5,
                      DONE => #DONE,
                      ERROR => #ERROR_MASTER_5,
                      STATUS => #STATUS_MASTER_5);
   END_IF;
   IF #_w1 AND #MODBUS_MASTER.ERROR THEN
       #ERROR_CODE := #MODBUS_MASTER.STATUS;
       #MASTER_DRIVER_LAST_ERROR := #INDEX_DRIVER;
   END_IF;
   IF #_w1 AND #MODBUS_MASTER.DONE AND (#INDEX_ADDR <> 4) THEN
       #ERROR_CODE := 0;
       #MASTER_DRIVER_LAST_ERROR := 0;
   END_IF;
   IF #_w1 AND #DONE THEN #DONE_PULSO := 1; END_IF;
END_REGION

REGION Network 2: Falha de comunicação Modbus
   // Conforme o cadastro em CICLE_TIMES_SET_ALARME, a comunicação Modbus irá acionar falha caso as tentativas excedam o cadastro. Caso a comunicação for bem sucedida, a falha irá resetar.
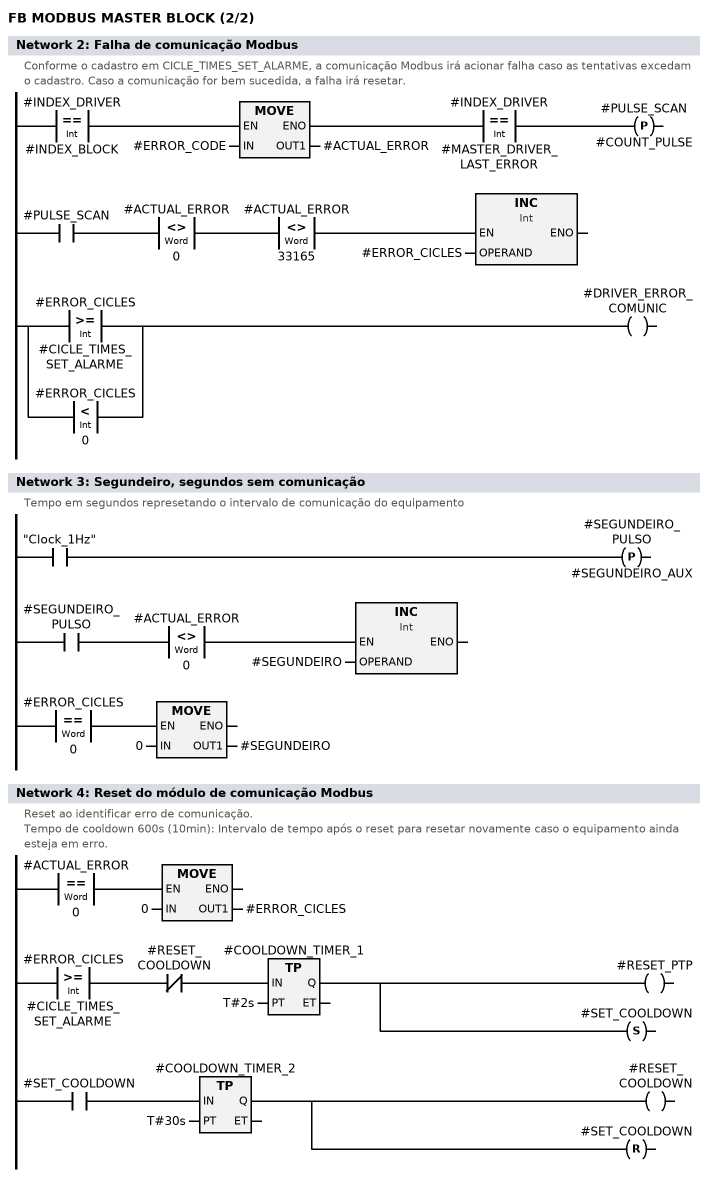
   #_w1 := #INDEX_DRIVER = #INDEX_BLOCK;
   IF #_w1 THEN #ACTUAL_ERROR := #ERROR_CODE; END_IF;
   #_w2 := #_w1 AND (#INDEX_DRIVER = #MASTER_DRIVER_LAST_ERROR);
   #PULSE_SCAN := #_w2 AND NOT #COUNT_PULSE;   // rising edge
   #COUNT_PULSE := #_w2;
   IF #PULSE_SCAN AND (#ACTUAL_ERROR <> 0) AND (#ACTUAL_ERROR <> 33165) THEN
       #ERROR_CICLES := #ERROR_CICLES + 1;
   END_IF;
   #DRIVER_ERROR_COMUNIC := (#ERROR_CICLES >= #CICLE_TIMES_SET_ALARME) OR (#ERROR_CICLES < 0);
END_REGION

REGION Network 3: Segundeiro, segundos sem comunicação
   // Tempo em segundos represetando o intervalo de comunicação do equipamento
   #SEGUNDEIRO_PULSO := "Clock_1Hz" AND NOT #SEGUNDEIRO_AUX;   // rising edge
   #SEGUNDEIRO_AUX := "Clock_1Hz";
   IF #SEGUNDEIRO_PULSO AND (#ACTUAL_ERROR <> 0) THEN #SEGUNDEIRO := #SEGUNDEIRO + 1; END_IF;
   IF #ERROR_CICLES = 0 THEN #SEGUNDEIRO := 0; END_IF;
END_REGION

REGION Network 4: Reset do módulo de comunicação Modbus
   // Reset ao identificar erro de comunicação.
   // Tempo de cooldown 600s (10min): Intervalo de tempo após o reset para resetar novamente caso o equipamento ainda esteja em erro.
   IF #ACTUAL_ERROR = 0 THEN #ERROR_CICLES := 0; END_IF;
   #COOLDOWN_TIMER_1.TP(IN := (#ERROR_CICLES >= #CICLE_TIMES_SET_ALARME) AND NOT #RESET_COOLDOWN, PT := T#2s);
   #RESET_PTP := #COOLDOWN_TIMER_1.Q;
   IF #COOLDOWN_TIMER_1.Q THEN #SET_COOLDOWN := TRUE; END_IF;
   #COOLDOWN_TIMER_2.TP(IN := #SET_COOLDOWN, PT := T#30s);
   #RESET_COOLDOWN := #COOLDOWN_TIMER_2.Q;
   IF #COOLDOWN_TIMER_2.Q THEN #SET_COOLDOWN := FALSE; END_IF;
END_REGION
END_FUNCTION_BLOCK

FUNCTION_BLOCK "FB MODBUS SCAN DRIVERS V2"   // FB30, LAD
TITLE = Function Block MODBUS SCAN DRIVERS: Varredura de drivers
{ S7_Optimized_Access := 'TRUE' }
VERSION : 0.1
   VAR_INPUT
      DONE : Bool;
      ERROR : Bool;
      QTD_DRIVER : Int;
      ID_START_DRIVER : Int;
      TAG_Nº_DRIVER : Int;
      IS_MMW_1 : Bool;
      ID_MMW_1 : Int;
      TAG_Nº_MMW_1 : Int;
      IS_MMW_2 : Bool;
      ID_MMW_2 : Int;
      TAG_Nº_MMW_2 : Int;
      IS_MMW_3 : Bool;
      ID_MMW_3 : Int;
      TAG_Nº_MMW_3 : Int;
      IS_MMW_4 : Bool;
      ID_MMW_4 : Int;
      TAG_Nº_MMW_4 : Int;
      UPDATE_TIME : Time;
   END_VAR
   VAR_OUTPUT
      MODBUS_ID : Int;
      INDEX_ADDR : Int;
      INDEX_DRIVER : Int;
      TRIGGER : Bool;
   END_VAR
   VAR
      CHANGE_DRIVER : Bool;
      AUX_CHANGE : Bool;
      AUX_FINISH : Bool;
      AUX1 : Bool;
      AUX2 : Bool;
      AUX3 : Bool;
      TAGS : Int := 3;
      "Timer" : IEC_TIMER;
      Timer_2 : IEC_TIMER;
   END_VAR
   VAR_TEMP   // added for the SCL form of the ladder/FBD networks
      _w1 : Bool;
      _w2 : Bool;
      _w3 : Bool;
      _w4 : Bool;
      _w5 : Bool;
      _w6 : Bool;
   END_VAR
BEGIN

REGION Network 1: Geração de variáveis para controle da varredura em "malha fechada"
   // Controle de malha fechado do Bloco modbus_Master.
   // O mesmo só pode ser chamado uma vez por módulo, ou seja necessita que seja multiplexado para atender mais de um escravo.
   // Para a lógica é usado um contato TOF, para controle do intervelo de tempo em que deve ser agregado o valor no INDEX(indice).
   // Após o telegrama ser encaminhado, sendo ele "True" ou "False" para DONE. O mesmo irá realimentar a malha de controle para que o próximo escravo seja chamado.
   // A situação acontece de igual forma para ERROR.
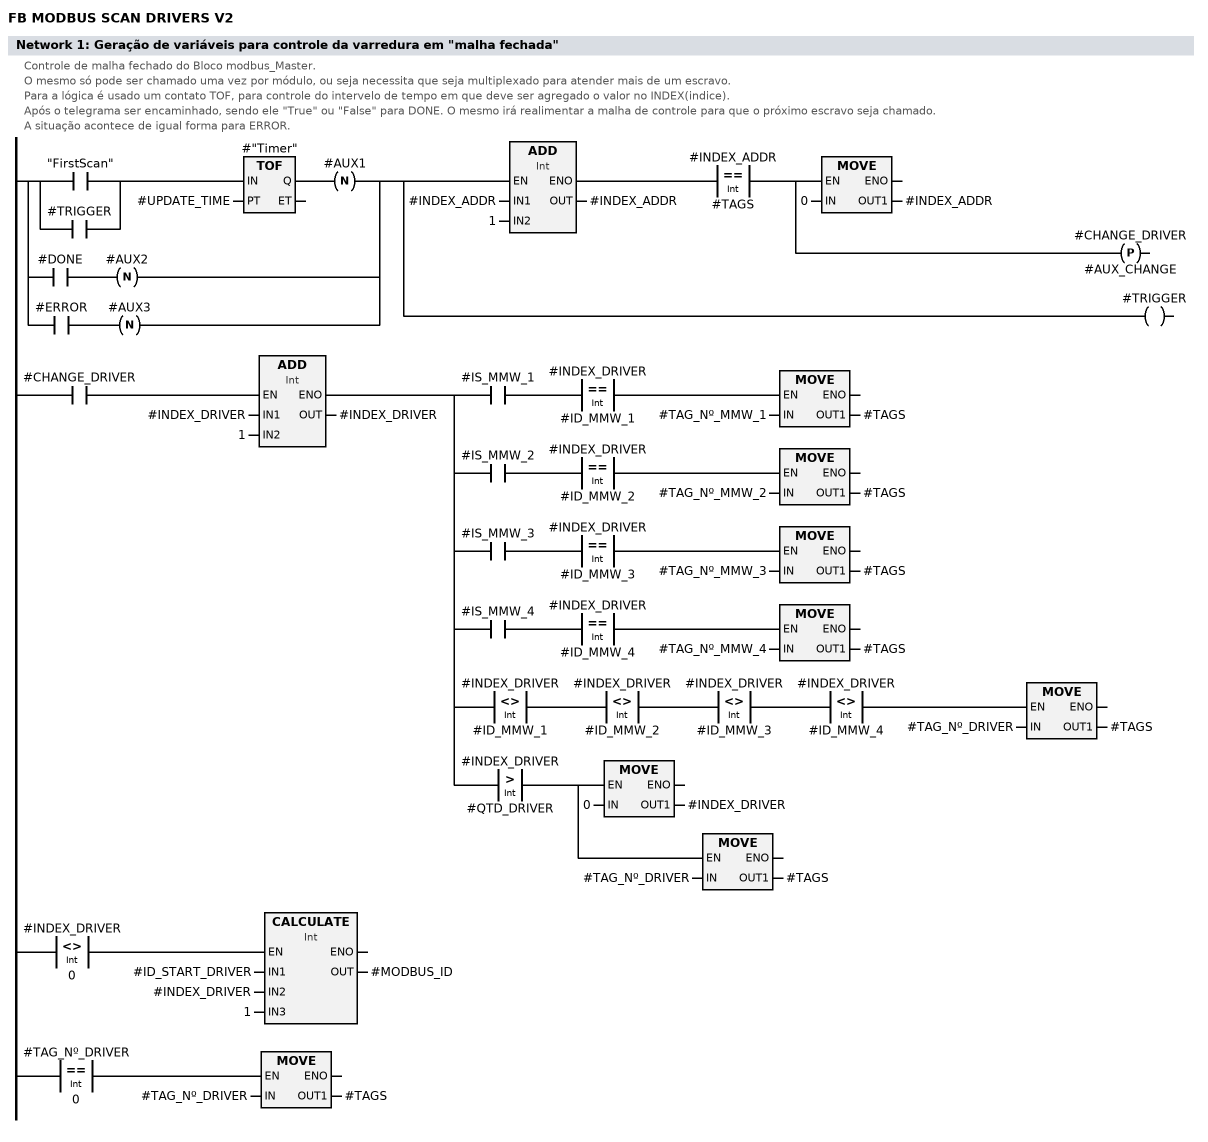
   #"Timer".TOF(IN := "FirstScan" OR #TRIGGER, PT := #UPDATE_TIME);
   #_w1 := NOT #"Timer".Q AND #AUX1;   // falling edge
   #AUX1 := #"Timer".Q;
   #_w2 := NOT #DONE AND #AUX2;   // falling edge
   #AUX2 := #DONE;
   #_w3 := NOT #ERROR AND #AUX3;   // falling edge
   #AUX3 := #ERROR;
   #_w4 := #_w1 OR #_w2 OR #_w3;
   IF #_w4 THEN #INDEX_ADDR := #INDEX_ADDR + 1; END_IF;
   #_w5 := #_w4 AND (#INDEX_ADDR = #TAGS);
   IF #_w5 THEN #INDEX_ADDR := 0; END_IF;
   #CHANGE_DRIVER := #_w5 AND NOT #AUX_CHANGE;   // rising edge
   #AUX_CHANGE := #_w5;
   #TRIGGER := #_w4;
   IF #CHANGE_DRIVER THEN #INDEX_DRIVER := #INDEX_DRIVER + 1; END_IF;
   IF #CHANGE_DRIVER AND #IS_MMW_1 AND (#INDEX_DRIVER = #ID_MMW_1) THEN #TAGS := #TAG_Nº_MMW_1; END_IF;
   IF #CHANGE_DRIVER AND #IS_MMW_2 AND (#INDEX_DRIVER = #ID_MMW_2) THEN #TAGS := #TAG_Nº_MMW_2; END_IF;
   IF #CHANGE_DRIVER AND #IS_MMW_3 AND (#INDEX_DRIVER = #ID_MMW_3) THEN #TAGS := #TAG_Nº_MMW_3; END_IF;
   IF #CHANGE_DRIVER AND #IS_MMW_4 AND (#INDEX_DRIVER = #ID_MMW_4) THEN #TAGS := #TAG_Nº_MMW_4; END_IF;
   IF #CHANGE_DRIVER AND (#INDEX_DRIVER <> #ID_MMW_1) AND (#INDEX_DRIVER <> #ID_MMW_2) AND (#INDEX_DRIVER <> #ID_MMW_3) AND (#INDEX_DRIVER <> #ID_MMW_4) THEN
       #TAGS := #TAG_Nº_DRIVER;
   END_IF;
   #_w6 := #CHANGE_DRIVER AND (#INDEX_DRIVER > #QTD_DRIVER);
   IF #_w6 THEN
       #INDEX_DRIVER := 0;
       #TAGS := #TAG_Nº_DRIVER;
   END_IF;
   IF #INDEX_DRIVER <> 0 THEN #MODBUS_ID := #ID_START_DRIVER + #INDEX_DRIVER - 1; END_IF;
   IF #TAG_Nº_DRIVER = 0 THEN #TAGS := #TAG_Nº_DRIVER; END_IF;
END_REGION
END_FUNCTION_BLOCK

FUNCTION_BLOCK "FB MODBUS SCAN DRIVERS V1"   // FB32, LAD
TITLE = Function Block MODBUS SCAN DRIVERS: Varredura de drivers
{ S7_Optimized_Access := 'TRUE' }
VERSION : 0.1
   VAR_INPUT
      DONE : Bool;
      ERROR : Bool;
      QTD_DRIVER : Int;
      ID_START_DRIVER : Int;
      IS_MMW : Bool;
      TAG_Nº_DRIVER : Int;
      TAG_Nº_MMW : Int;
      UPDATE_TIME : Time;
   END_VAR
   VAR_OUTPUT
      MODBUS_ID : Int;
      INDEX_ADDR : Int;
      INDEX_DRIVER : Int;
      TRIGGER : Bool;
   END_VAR
   VAR
      CHANGE_DRIVER : Bool;
      AUX_CHANGE : Bool;
      AUX_FINISH : Bool;
      AUX1 : Bool;
      AUX2 : Bool;
      AUX3 : Bool;
      TAGS : Int := 3;
      "Timer" : IEC_TIMER;
      Timer_2 : IEC_TIMER;
   END_VAR
   VAR_TEMP   // added for the SCL form of the ladder/FBD networks
      _w1 : Bool;
      _w2 : Bool;
      _w3 : Bool;
      _w4 : Bool;
      _w5 : Bool;
      _w6 : Bool;
   END_VAR
BEGIN

REGION Network 1: Geração de variáveis para controle da varredura em "malha fechada"
   // Controle de malha fechado do Bloco modbus_Master.
   // O mesmo só pode ser chamado uma vez por módulo, ou seja necessita que seja multiplexado para atender mais de um escravo.
   // Para a lógica é usado um contato TOF, para controle do intervelo de tempo em que deve ser agregado o valor no INDEX(indice).
   // Após o telegrama ser encaminhado, sendo ele "True" ou "False" para DONE. O mesmo irá realimentar a malha de controle para que o próximo escravo seja chamado.
   // A situação acontece de igual forma para ERROR.
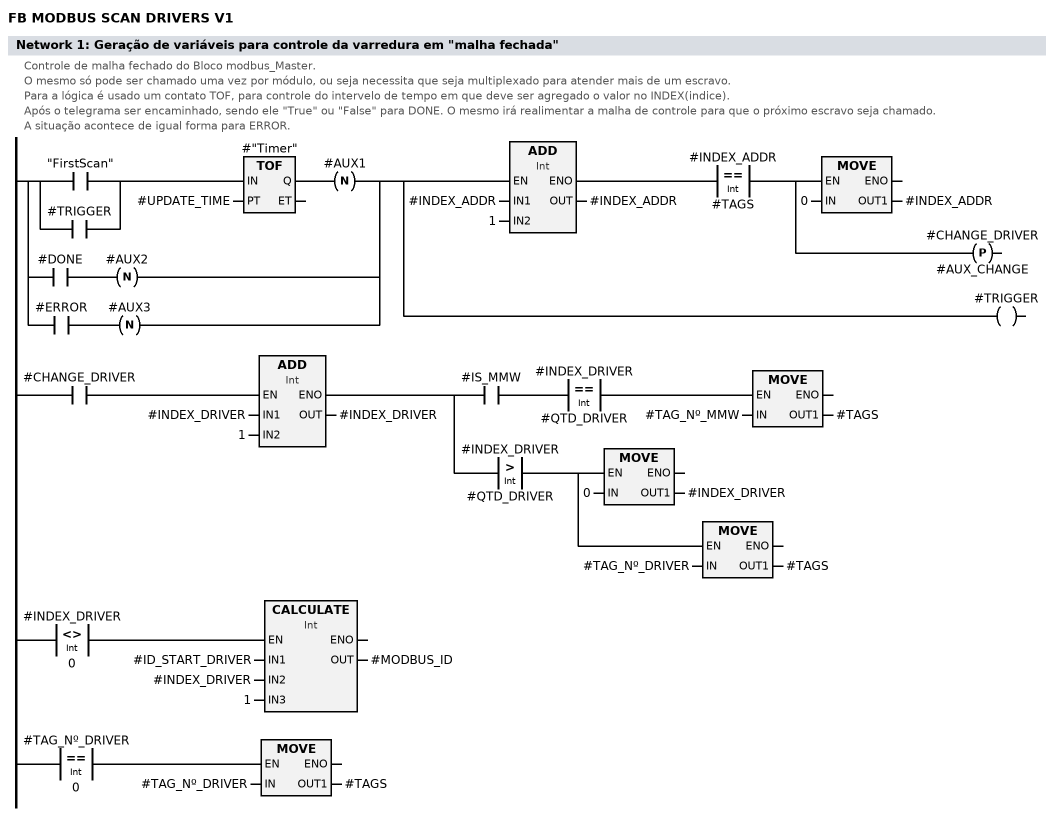
   #"Timer".TOF(IN := "FirstScan" OR #TRIGGER, PT := #UPDATE_TIME);
   #_w1 := NOT #"Timer".Q AND #AUX1;   // falling edge
   #AUX1 := #"Timer".Q;
   #_w2 := NOT #DONE AND #AUX2;   // falling edge
   #AUX2 := #DONE;
   #_w3 := NOT #ERROR AND #AUX3;   // falling edge
   #AUX3 := #ERROR;
   #_w4 := #_w1 OR #_w2 OR #_w3;
   IF #_w4 THEN #INDEX_ADDR := #INDEX_ADDR + 1; END_IF;
   #_w5 := #_w4 AND (#INDEX_ADDR = #TAGS);
   IF #_w5 THEN #INDEX_ADDR := 0; END_IF;
   #CHANGE_DRIVER := #_w5 AND NOT #AUX_CHANGE;   // rising edge
   #AUX_CHANGE := #_w5;
   #TRIGGER := #_w4;
   IF #CHANGE_DRIVER THEN #INDEX_DRIVER := #INDEX_DRIVER + 1; END_IF;
   IF #CHANGE_DRIVER AND #IS_MMW AND (#INDEX_DRIVER = #QTD_DRIVER) THEN #TAGS := #TAG_Nº_MMW; END_IF;
   #_w6 := #CHANGE_DRIVER AND (#INDEX_DRIVER > #QTD_DRIVER);
   IF #_w6 THEN
       #INDEX_DRIVER := 0;
       #TAGS := #TAG_Nº_DRIVER;
   END_IF;
   IF #INDEX_DRIVER <> 0 THEN #MODBUS_ID := #ID_START_DRIVER + #INDEX_DRIVER - 1; END_IF;
   IF #TAG_Nº_DRIVER = 0 THEN #TAGS := #TAG_Nº_DRIVER; END_IF;
END_REGION
END_FUNCTION_BLOCK

// ===== library: MasterCopy "1.1 Acionamento" =====

// folder: 1. FB Bilbiotecas/1.1 Acionamento

FUNCTION_BLOCK "FB CONDIÇÃO DE PARTIDA"   // FB6, LAD
TITLE = Function Block CONDIÇÃO DE PARTIDA - Intertravamentos para partir o motor/bomba
{ S7_Optimized_Access := 'TRUE' }
VERSION : 0.1
// Network 1: Gerenciamento Status Motor/Bomba
// Network 2: Recebimento dos sinais de entrada (Sinais de campo e comandos)
// Network 3: MODO MANUAL: Conjunto de condições para ligar e desligar
// Network 4: MODO AUTOMÁTICO: Conjunto de condições para ligar e desligar
// Network 5: FALHA: Condicionamento de falha
// Network 6: LIGA BOMBA: Validando intertravamentos para ligar
   VAR_INPUT
      INPUT_LIGADO : Bool;   // 1 = Sinal elétrico de campo indicando bomba ligada
      INPUT_DESLIGADO : Bool;   // 1 = Sinal elétrico de campo indicando bomba desligada
      INPUT_FALHA : Bool;   // 0 = Sinal elétrico de campo indicando bomba em falha
      INPUT_LOCAL_MAN : Bool;   // 1 = Sinal elétrico de campo indicando bomba em local
      INPUT_LOCAL_AUTO : Bool;   // 1 = Sinal elétrico de campo indicando bomba em local automático
      INPUT_REMOTO : Bool;   // 1 = Sinal elétrico de campo indicando bomba em remoto
      INPUT_FALHA_PROFINET : Bool;   // 1 = Indica falta de comunicação PROFINET com o equipamento
      INPUT_HABILITA_LIGA_AUTO : Bool;   // 1 = Sinal para habilitar Liga Bomba em Modo Automático quando todas as condições foram atentidas
      INPUT_CMD_LIGA : Bool;   // Comando enviado da IHM/SCADA para ligar a bomba
      CMD_MANUTEN : Bool;   // Comando enviado da IHM/SCADA para colocar a bomba em Modo de Manutenção
      CMD_MODO_OPERACAO : Bool;   // Comando enviado da IHM/SCADA para colocar a bomba em (0 = Modo Manual, 1 = Modo Automático)
      CMD_RESET_HORIMETRO : Bool;
   END_VAR
   VAR_OUTPUT
      LIGA_BOMBA : Bool;   // Saída acionada para ligar a bomba remotamente
      STATUS_MOTOR : Byte;   // 0 = DESLIGADO; 1 = LIGADO; 2 = FALHA; 3 = MANUTENÇÃO; 4 = SEM COMUNICAÇÃO MODBUS
      OUTPUT_REMOTO_AUTO : Bool;   // Saída para indicar bomba em Remoto Automático
      OUTPUT_MODO_OPER : Byte;
      STS_HORIMETRO : UInt;
      RESET_CMD_LIGA : Bool;
      STS_INTERTRAVAMENTO_AUTOMATICO : Bool;
   END_VAR
   VAR
      LOCAL_MAN : Bool;   // Saída para indicar bomba em Local Manual
      REMOTO_MAN : Bool;   // Saída para indicar bomba em Remoto Manual
      MANUTEN : Bool;   // Variável local para Indicar bomba em Modo Manutenção
      REMOTO : Bool;   // Variável local para indicar bomba em Modo Remoto
      FALHA : Bool;   // Variável local para indicar bomba em Falha
      LOCAL_AUTO : Bool;   // Variável local para indicar bomba em Modo Local Automático
      LIGA_REM_MAN : Bool;   // Variável local para Acionamento Remoto Manual
      LIGA_REM_AUTO : Bool;   // Variável local para Acionamento Remoto Automático
      "FB MODOS DE OPERAÇÃO_Instance" : "FB MODOS DE OPERAÇÃO";
      FB_HORÍMETRO_Instance : "FB_HORÍMETRO";
   END_VAR
   VAR_TEMP   // added for the SCL form of the ladder/FBD networks
      _w1 : Bool;
   END_VAR
BEGIN

REGION Network 1: Recebimento dos sinais de entrada (Sinais de campo e comandos)
   // INPUT_ABERTA = Entrada de sinal de Bomba Ligada
   // INPUT_FECHADA = Entrada de sinal de Bomba Desligada
   // INPUT_FALHA = Entrada de sinal de Bomba em Falha
   // INPUT_FALHA_PROFINET = Sem comunicação Profinet
   // STATUS_MOTOR: 0 = DESLIGADO; 1 = LIGADO; 2 = FALHA; 3 = MANUTENÇÃO; 4 = SEM COMUNICAÇÃO MODBUS
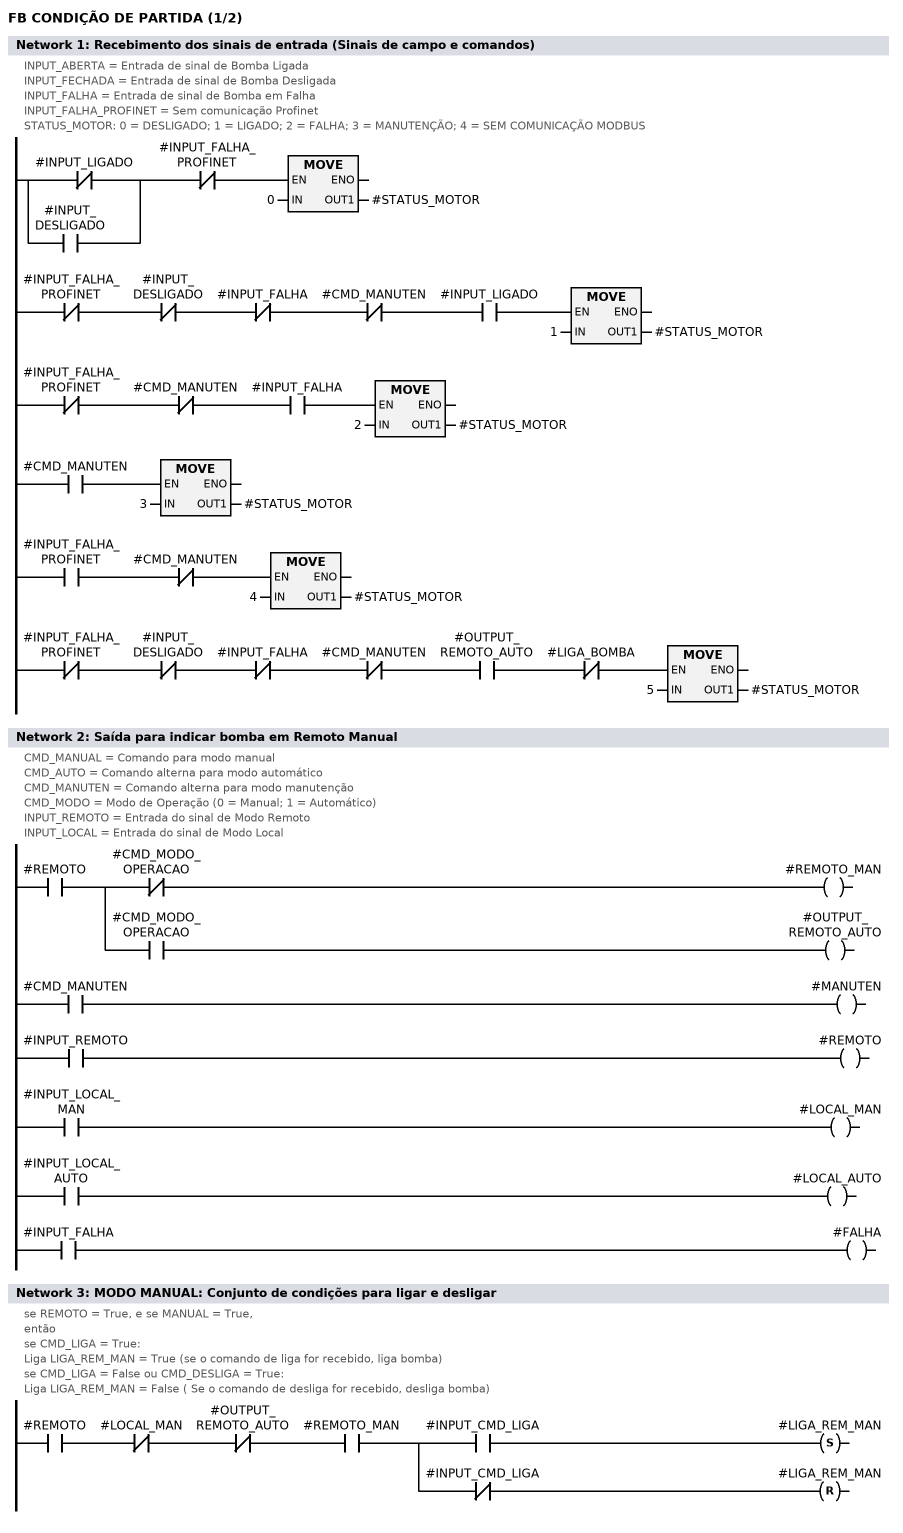
   RUNG wire#powerrail
      I_Contact( #INPUT_LIGADO )
      wire#w1
      I_Contact( #INPUT_FALHA_PROFINET )
      Move(in := 0, out1 => #STATUS_MOTOR)
   END_RUNG
   RUNG wire#powerrail
      Contact( #INPUT_DESLIGADO )
   END_RUNG wire#w1
   RUNG wire#powerrail
      I_Contact( #INPUT_FALHA_PROFINET )
      I_Contact( #INPUT_DESLIGADO )
      I_Contact( #INPUT_FALHA )
      I_Contact( #CMD_MANUTEN )
      Contact( #INPUT_LIGADO )
      Move(in := 1, out1 => #STATUS_MOTOR)
   END_RUNG
   RUNG wire#powerrail
      I_Contact( #INPUT_FALHA_PROFINET )
      I_Contact( #CMD_MANUTEN )
      Contact( #INPUT_FALHA )
      Move(in := 2, out1 => #STATUS_MOTOR)
   END_RUNG
   RUNG wire#powerrail
      Contact( #CMD_MANUTEN )
      Move(in := 3, out1 => #STATUS_MOTOR)
   END_RUNG
   RUNG wire#powerrail
      Contact( #INPUT_FALHA_PROFINET )
      I_Contact( #CMD_MANUTEN )
      Move(in := 4, out1 => #STATUS_MOTOR)
   END_RUNG
   RUNG wire#powerrail
      I_Contact( #INPUT_FALHA_PROFINET )
      I_Contact( #INPUT_DESLIGADO )
      I_Contact( #INPUT_FALHA )
      I_Contact( #CMD_MANUTEN )
      Contact( #OUTPUT_REMOTO_AUTO )
      I_Contact( #LIGA_BOMBA )
      Move(in := 5, out1 => #STATUS_MOTOR)
   END_RUNG
   // the same network as SCL:
   IF (NOT #INPUT_LIGADO OR #INPUT_DESLIGADO) AND NOT #INPUT_FALHA_PROFINET THEN #STATUS_MOTOR := 0; END_IF;
   IF NOT #INPUT_FALHA_PROFINET AND NOT #INPUT_DESLIGADO AND NOT #INPUT_FALHA AND NOT #CMD_MANUTEN AND #INPUT_LIGADO THEN
       #STATUS_MOTOR := 1;
   END_IF;
   IF NOT #INPUT_FALHA_PROFINET AND NOT #CMD_MANUTEN AND #INPUT_FALHA THEN #STATUS_MOTOR := 2; END_IF;
   IF #CMD_MANUTEN THEN #STATUS_MOTOR := 3; END_IF;
   IF #INPUT_FALHA_PROFINET AND NOT #CMD_MANUTEN THEN #STATUS_MOTOR := 4; END_IF;
   IF NOT #INPUT_FALHA_PROFINET AND NOT #INPUT_DESLIGADO AND NOT #INPUT_FALHA AND NOT #CMD_MANUTEN AND #OUTPUT_REMOTO_AUTO AND NOT #LIGA_BOMBA THEN
       #STATUS_MOTOR := 5;
   END_IF;
END_REGION

REGION Network 2: Saída para indicar bomba em Remoto Manual
   // CMD_MANUAL = Comando para modo manual
   // CMD_AUTO = Comando alterna para modo automático
   // CMD_MANUTEN = Comando alterna para modo manutenção
   // CMD_MODO = Modo de Operação (0 = Manual; 1 = Automático)
   // INPUT_REMOTO = Entrada do sinal de Modo Remoto
   // INPUT_LOCAL = Entrada do sinal de Modo Local
   RUNG wire#powerrail
      Contact( #REMOTO )
      wire#w1
      I_Contact( #CMD_MODO_OPERACAO )
      Coil( #REMOTO_MAN )
   END_RUNG
   RUNG wire#w1
      Contact( #CMD_MODO_OPERACAO )
      Coil( #OUTPUT_REMOTO_AUTO )
   END_RUNG
   RUNG wire#powerrail
      Contact( #CMD_MANUTEN )
      Coil( #MANUTEN )
   END_RUNG
   RUNG wire#powerrail
      Contact( #INPUT_REMOTO )
      Coil( #REMOTO )
   END_RUNG
   RUNG wire#powerrail
      Contact( #INPUT_LOCAL_MAN )
      Coil( #LOCAL_MAN )
   END_RUNG
   RUNG wire#powerrail
      Contact( #INPUT_LOCAL_AUTO )
      Coil( #LOCAL_AUTO )
   END_RUNG
   RUNG wire#powerrail
      Contact( #INPUT_FALHA )
      Coil( #FALHA )
   END_RUNG
   // the same network as SCL:
   #REMOTO_MAN := #REMOTO AND NOT #CMD_MODO_OPERACAO;
   #OUTPUT_REMOTO_AUTO := #REMOTO AND #CMD_MODO_OPERACAO;
   #MANUTEN := #CMD_MANUTEN;
   #REMOTO := #INPUT_REMOTO;
   #LOCAL_MAN := #INPUT_LOCAL_MAN;
   #LOCAL_AUTO := #INPUT_LOCAL_AUTO;
   #FALHA := #INPUT_FALHA;
END_REGION

REGION Network 3: MODO MANUAL: Conjunto de condições para ligar e desligar
   // se REMOTO = True, e se MANUAL = True,
   // 
   // então
   // se CMD_LIGA = True: 
   // Liga LIGA_REM_MAN = True (se o comando de liga for recebido, liga bomba)
   // 
   // se CMD_LIGA = False ou CMD_DESLIGA = True:
   // Liga LIGA_REM_MAN = False ( Se o comando de desliga for recebido, desliga bomba)
   RUNG wire#powerrail
      Contact( #REMOTO )
      I_Contact( #LOCAL_MAN )
      I_Contact( #OUTPUT_REMOTO_AUTO )
      Contact( #REMOTO_MAN )
      wire#w1
      Contact( #INPUT_CMD_LIGA )
      S_Coil( #LIGA_REM_MAN )
   END_RUNG
   RUNG wire#w1
      I_Contact( #INPUT_CMD_LIGA )
      R_Coil( #LIGA_REM_MAN )
   END_RUNG
   // the same network as SCL:
   #_w1 := #REMOTO AND NOT #LOCAL_MAN AND NOT #OUTPUT_REMOTO_AUTO AND #REMOTO_MAN;
   IF #_w1 AND #INPUT_CMD_LIGA THEN #LIGA_REM_MAN := TRUE; END_IF;
   IF #_w1 AND NOT #INPUT_CMD_LIGA THEN #LIGA_REM_MAN := FALSE; END_IF;
END_REGION

REGION Network 4: Variável local para Acionamento Remoto Auto
   // se REMOTO = True, e se AUTO = True:
   // 
   // então
   // se LIGA_REM_AUTO = True:
   // e se PARAMETRO < PARAMETRO_LIGA;
   // então LIGA_REM_AUTO = True (se a leitura for menor que o cadastro para ligar, liga em remoto automático)
   // 
   // se LIGA_REM_AUTO = False:
   // e se PARAMETRO >= PARAMETRO_DESLIGA:
   // então Desliga REMOTO AUTOMÁTICO (se a leitura for maior ou igual ao cadastro para desligar, desliga em remoto automático)
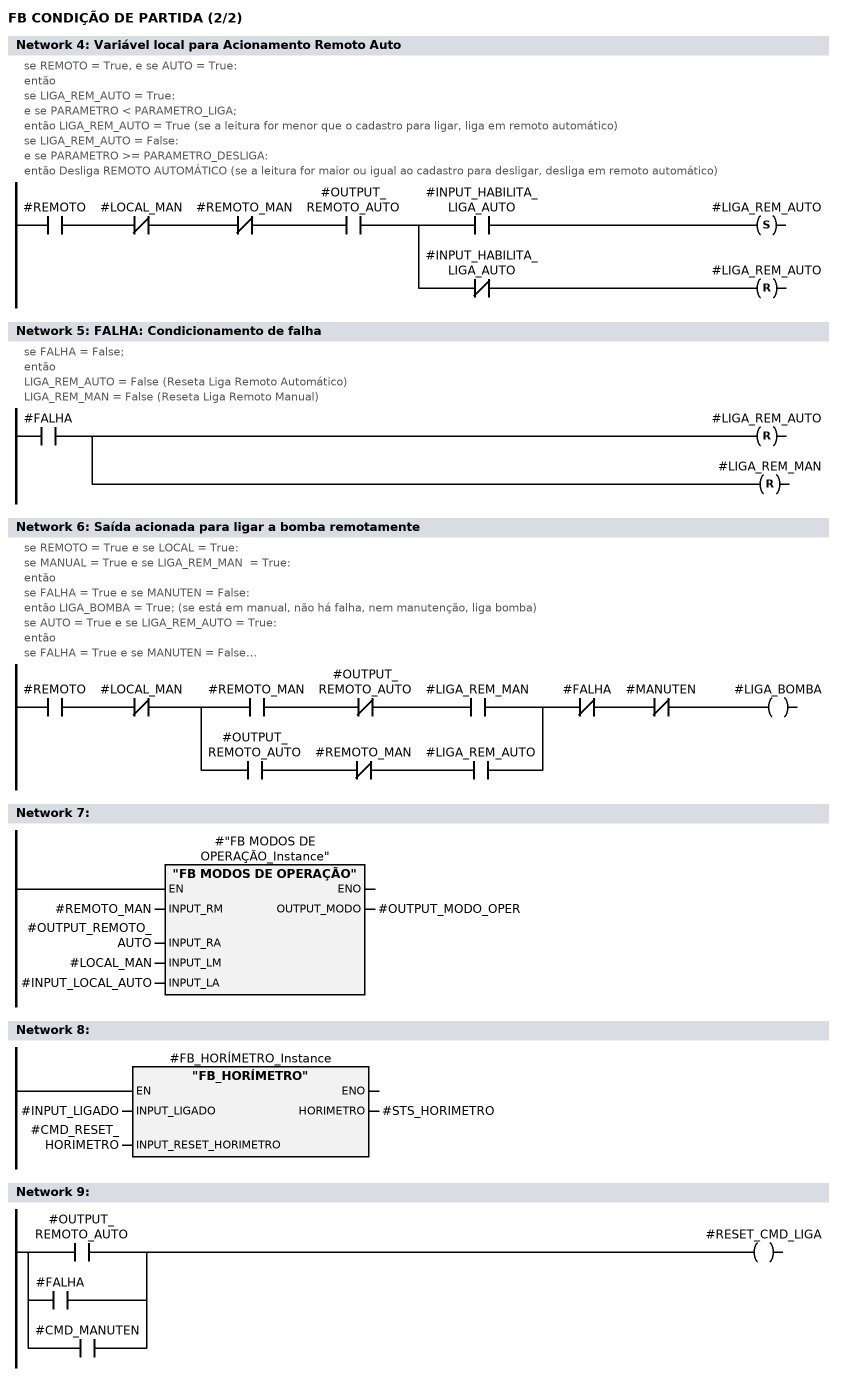
   RUNG wire#powerrail
      Contact( #REMOTO )
      I_Contact( #LOCAL_MAN )
      I_Contact( #REMOTO_MAN )
      Contact( #OUTPUT_REMOTO_AUTO )
      wire#w1
      Contact( #INPUT_HABILITA_LIGA_AUTO )
      S_Coil( #LIGA_REM_AUTO )
   END_RUNG
   RUNG wire#w1
      I_Contact( #INPUT_HABILITA_LIGA_AUTO )
      R_Coil( #LIGA_REM_AUTO )
   END_RUNG
   // the same network as SCL:
   #_w1 := #REMOTO AND NOT #LOCAL_MAN AND NOT #REMOTO_MAN AND #OUTPUT_REMOTO_AUTO;
   IF #_w1 AND #INPUT_HABILITA_LIGA_AUTO THEN #LIGA_REM_AUTO := TRUE; END_IF;
   IF #_w1 AND NOT #INPUT_HABILITA_LIGA_AUTO THEN #LIGA_REM_AUTO := FALSE; END_IF;
END_REGION

REGION Network 5: FALHA: Condicionamento de falha
   // se FALHA = False;
   // 
   // então
   // LIGA_REM_AUTO = False (Reseta Liga Remoto Automático)
   // LIGA_REM_MAN = False (Reseta Liga Remoto Manual)
   RUNG wire#powerrail
      Contact( #FALHA )
      wire#w1
      R_Coil( #LIGA_REM_AUTO )
   END_RUNG
   RUNG wire#w1
      R_Coil( #LIGA_REM_MAN )
   END_RUNG
   // the same network as SCL:
   IF #FALHA THEN
       #LIGA_REM_AUTO := FALSE;
       #LIGA_REM_MAN := FALSE;
   END_IF;
END_REGION

REGION Network 6: Saída acionada para ligar a bomba remotamente
   // se REMOTO = True e se LOCAL = True:
   // 
   // se MANUAL = True e se LIGA_REM_MAN  = True:
   // então
   // se FALHA = True e se MANUTEN = False:
   // então LIGA_BOMBA = True; (se está em manual, não há falha, nem manutenção, liga bomba)
   // 
   // se AUTO = True e se LIGA_REM_AUTO = True:
   // então
   // se FALHA = True e se MANUTEN = False:
   // então LIGA_BOMBA = True; (se está em automático, não há falha, nem manutenção, liga bomba)
   RUNG wire#powerrail
      Contact( #REMOTO )
      I_Contact( #LOCAL_MAN )
      wire#w1
      Contact( #REMOTO_MAN )
      I_Contact( #OUTPUT_REMOTO_AUTO )
      Contact( #LIGA_REM_MAN )
      wire#w2
      I_Contact( #FALHA )
      I_Contact( #MANUTEN )
      Coil( #LIGA_BOMBA )
   END_RUNG
   RUNG wire#w1
      Contact( #OUTPUT_REMOTO_AUTO )
      I_Contact( #REMOTO_MAN )
      Contact( #LIGA_REM_AUTO )
   END_RUNG wire#w2
   // the same network as SCL:
   #LIGA_BOMBA := #REMOTO AND NOT #LOCAL_MAN AND ((#REMOTO_MAN AND NOT #OUTPUT_REMOTO_AUTO AND #LIGA_REM_MAN) OR (#OUTPUT_REMOTO_AUTO AND NOT #REMOTO_MAN AND #LIGA_REM_AUTO)) AND NOT #FALHA AND NOT #MANUTEN;
END_REGION

REGION Network 7
   RUNG wire#powerrail
      #"FB MODOS DE OPERAÇÃO_Instance"(INPUT_RM := #REMOTO_MAN, INPUT_RA := #OUTPUT_REMOTO_AUTO, INPUT_LM := #LOCAL_MAN, INPUT_LA := #INPUT_LOCAL_AUTO, OUTPUT_MODO => #OUTPUT_MODO_OPER)
   END_RUNG
   // the same network as SCL:
   #"FB MODOS DE OPERAÇÃO_Instance"(INPUT_RM := #REMOTO_MAN,   // "FB MODOS DE OPERAÇÃO"
                           INPUT_RA := #OUTPUT_REMOTO_AUTO,
                           INPUT_LM := #LOCAL_MAN,
                           INPUT_LA := #INPUT_LOCAL_AUTO,
                           OUTPUT_MODO => #OUTPUT_MODO_OPER);
END_REGION

REGION Network 8
   RUNG wire#powerrail
      #FB_HORÍMETRO_Instance(INPUT_LIGADO := #INPUT_LIGADO, INPUT_RESET_HORIMETRO := #CMD_RESET_HORIMETRO, HORIMETRO => #STS_HORIMETRO)
   END_RUNG
   // the same network as SCL:
   #FB_HORÍMETRO_Instance(INPUT_LIGADO := #INPUT_LIGADO,   // "FB_HORÍMETRO"
                          INPUT_RESET_HORIMETRO := #CMD_RESET_HORIMETRO,
                          HORIMETRO => #STS_HORIMETRO);
END_REGION

REGION Network 9
   RUNG wire#powerrail
      Contact( #OUTPUT_REMOTO_AUTO )
      wire#w1
      Coil( #RESET_CMD_LIGA )
   END_RUNG
   RUNG wire#powerrail
      Contact( #FALHA )
   END_RUNG wire#w1
   RUNG wire#powerrail
      Contact( #CMD_MANUTEN )
   END_RUNG wire#w1
   // the same network as SCL:
   #RESET_CMD_LIGA := #OUTPUT_REMOTO_AUTO OR #FALHA OR #CMD_MANUTEN;
END_REGION
END_FUNCTION_BLOCK

FUNCTION_BLOCK "FB_LIGA/DESLIGA MODO AUTO"   // FB8, LAD
TITLE = Function Block LIGA/DESLIGA MODO AUTO
{ S7_Optimized_Access := 'TRUE' }
VERSION : 0.1
// Bloco para alternância dinâmica do tempo para ligar e desligar bomba.
// Network 1: Atribuição do sinal de liga
// Network 2: Function Block CONTADOR: Contador de tempo para bomba ligada
// Network 3: Comparativo de bomba ligada com tempo cadastrado para ficar ligada
// Network 4: Function Block CONTADOR: Contador de tempo para bomba desligada
// Network 5: Comparativo de bomba desligada com tempo cadastrado para ficar desligada
// Network 6: Transferindo sinal de bomba ligada/desligada para fora do bloco
   VAR_INPUT
      REMOTO_AUTO : Bool;   // Modo Remoto Automático
      CAD_TEMPO_LIGADA : Real;   // Cadastro tempo para bomba ficar ligada
      CAD_TEMPO_DESLIGADA : Real;   // Cadastro tempo para bomba ficar desligada
      TEMPO_ALTERNANCIA : Bool;   // Controle de alternancia entre bombas
   END_VAR
   VAR_OUTPUT
      HABILITA_LIGA_AUTO : Bool;   // Habilita Liga em Modo Automático
   END_VAR
   VAR_IN_OUT
      TEMPO_LIGADA_AUTO_SEG : Real;   // Tempo de bomba ligada em Modo Automático (segundos)
      TEMPO_LIGADA_AUTO_MIN : Real;   // Tempo de bomba ligada em Modo Automático (minutos)
      TEMPO_LIGADA_AUTO_HOR : Real;   // Tempo de bomba ligada em Modo Automático (horas)
      TEMPO_DESLIGADA_AUTO_SEG : Real;   // Tempo de bomba desligada em Modo Automático (segundos)
      TEMPO_DESLIGADA_AUTO_MIN : Real;   // Tempo de bomba desligada em Modo Automático (minutos)
      TEMPO_DESLIGADA_AUTO_HOR : Real;   // Tempo de bomba desligada em Modo Automático (horas)
   END_VAR
   VAR
      DESLIGA_AUTO : Bool;   // Desliga bomba em Modo Automático
      LIGA_AUTO : Bool;   // Liga bomba em Modo Automático
      MINUTEIRO_LIGADA : "FB CONTADOR";
      MINUTEIRO_DESLIGADA : "FB CONTADOR";
      TEMPO_LIGADA_AUTO_HORA : Bool;   // Tempo de bomba desligada em Modo Automático (em horas)
   END_VAR
BEGIN

REGION Network 1: Atribuição do sinal de liga
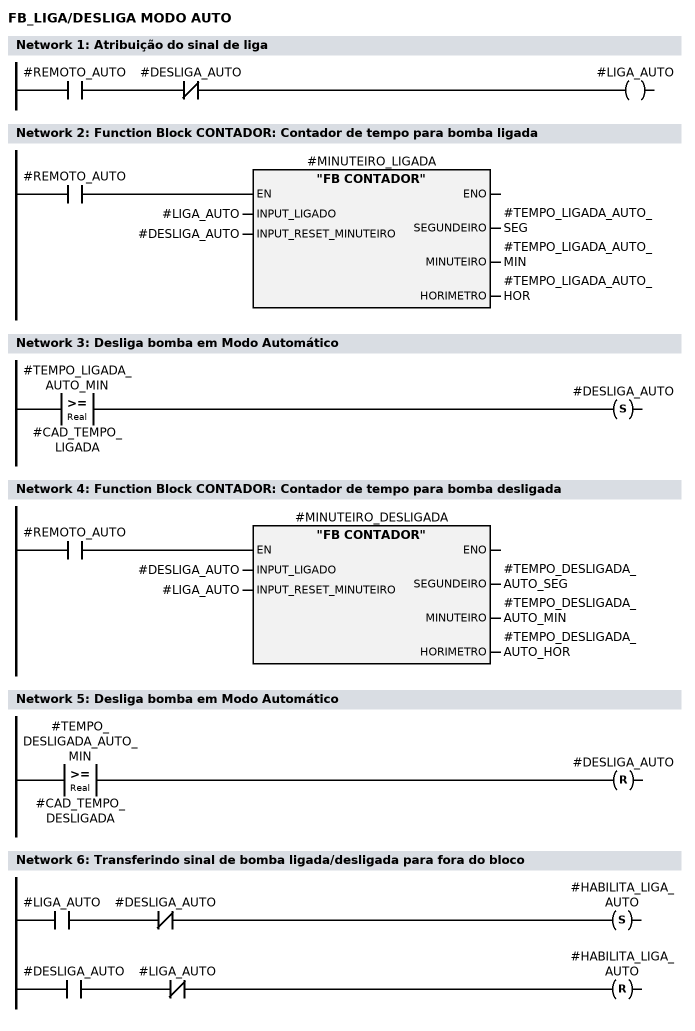
   RUNG wire#powerrail
      Contact( #REMOTO_AUTO )
      I_Contact( #DESLIGA_AUTO )
      Coil( #LIGA_AUTO )
   END_RUNG
   // the same network as SCL:
   #LIGA_AUTO := #REMOTO_AUTO AND NOT #DESLIGA_AUTO;
END_REGION

REGION Network 2: Function Block CONTADOR: Contador de tempo para bomba ligada
   RUNG wire#powerrail
      Contact( #REMOTO_AUTO )
      #MINUTEIRO_LIGADA(INPUT_LIGADO := #LIGA_AUTO, INPUT_RESET_MINUTEIRO := #DESLIGA_AUTO, SEGUNDEIRO => #TEMPO_LIGADA_AUTO_SEG, MINUTEIRO => #TEMPO_LIGADA_AUTO_MIN, HORIMETRO => #TEMPO_LIGADA_AUTO_HOR)
   END_RUNG
   // the same network as SCL:
   IF #REMOTO_AUTO THEN
       #MINUTEIRO_LIGADA(INPUT_LIGADO := #LIGA_AUTO,   // "FB CONTADOR"
                         INPUT_RESET_MINUTEIRO := #DESLIGA_AUTO,
                         SEGUNDEIRO => #TEMPO_LIGADA_AUTO_SEG,
                         MINUTEIRO => #TEMPO_LIGADA_AUTO_MIN,
                         HORIMETRO => #TEMPO_LIGADA_AUTO_HOR);
   END_IF;
END_REGION

REGION Network 3: Desliga bomba em Modo Automático
   RUNG wire#powerrail
      { S7_Templates := "SrcType := Real" } GE_Contact(in1 := #TEMPO_LIGADA_AUTO_MIN, in2 := #CAD_TEMPO_LIGADA)
      S_Coil( #DESLIGA_AUTO )
   END_RUNG
   // the same network as SCL:
   IF #TEMPO_LIGADA_AUTO_MIN >= #CAD_TEMPO_LIGADA THEN #DESLIGA_AUTO := TRUE; END_IF;
END_REGION

REGION Network 4: Function Block CONTADOR: Contador de tempo para bomba desligada
   RUNG wire#powerrail
      Contact( #REMOTO_AUTO )
      #MINUTEIRO_DESLIGADA(INPUT_LIGADO := #DESLIGA_AUTO, INPUT_RESET_MINUTEIRO := #LIGA_AUTO, SEGUNDEIRO => #TEMPO_DESLIGADA_AUTO_SEG, MINUTEIRO => #TEMPO_DESLIGADA_AUTO_MIN, HORIMETRO => #TEMPO_DESLIGADA_AUTO_HOR)
   END_RUNG
   // the same network as SCL:
   IF #REMOTO_AUTO THEN
       #MINUTEIRO_DESLIGADA(INPUT_LIGADO := #DESLIGA_AUTO,   // "FB CONTADOR"
                            INPUT_RESET_MINUTEIRO := #LIGA_AUTO,
                            SEGUNDEIRO => #TEMPO_DESLIGADA_AUTO_SEG,
                            MINUTEIRO => #TEMPO_DESLIGADA_AUTO_MIN,
                            HORIMETRO => #TEMPO_DESLIGADA_AUTO_HOR);
   END_IF;
END_REGION

REGION Network 5: Desliga bomba em Modo Automático
   RUNG wire#powerrail
      { S7_Templates := "SrcType := Real" } GE_Contact(in1 := #TEMPO_DESLIGADA_AUTO_MIN, in2 := #CAD_TEMPO_DESLIGADA)
      R_Coil( #DESLIGA_AUTO )
   END_RUNG
   // the same network as SCL:
   IF #TEMPO_DESLIGADA_AUTO_MIN >= #CAD_TEMPO_DESLIGADA THEN #DESLIGA_AUTO := FALSE; END_IF;
END_REGION

REGION Network 6: Transferindo sinal de bomba ligada/desligada para fora do bloco
   RUNG wire#powerrail
      Contact( #LIGA_AUTO )
      I_Contact( #DESLIGA_AUTO )
      S_Coil( #HABILITA_LIGA_AUTO )
   END_RUNG
   RUNG wire#powerrail
      Contact( #DESLIGA_AUTO )
      I_Contact( #LIGA_AUTO )
      R_Coil( #HABILITA_LIGA_AUTO )
   END_RUNG
   // the same network as SCL:
   IF #LIGA_AUTO AND NOT #DESLIGA_AUTO THEN #HABILITA_LIGA_AUTO := TRUE; END_IF;
   IF #DESLIGA_AUTO AND NOT #LIGA_AUTO THEN #HABILITA_LIGA_AUTO := FALSE; END_IF;
END_REGION
END_FUNCTION_BLOCK

FUNCTION_BLOCK "FB MODOS DE OPERAÇÃO"   // FB10, LAD
TITLE = Function Block MODOS DE OPERAÇÃO
{ S7_Optimized_Access := 'TRUE' }
VERSION : 0.1
// Movendo os valores booleados para uma variável do tipo int
   VAR_INPUT
      INPUT_RM : Bool;   // Entrada de sinal alto para indicar modo Remoto Manual
      INPUT_RA : Bool;   // Entrada de sinal alto para indicar modo Remoto Automático
      INPUT_LM : Bool;   // Entrada de sinal alto para indicar modo Local Manual
      INPUT_LA : Bool;   // Entrada de sinal alto para indicar modo Local Automático
   END_VAR
   VAR_OUTPUT
      OUTPUT_MODO : Int;   // Saída do Modo de Operação
   END_VAR
BEGIN

REGION Network 1: Estrutura de Operação
   // Se Remoto Manual = TRUE, OPERACAO_MOTOR = 1 
   // Se Remoto Automático = TRUE, OPERACAO_MOTOR = 2
   // Se Local Automático = TRUE, OPERACAO_MOTOR = 3
   // Se Local Manual = TRUE, OPERACAO_MOTOR = 4
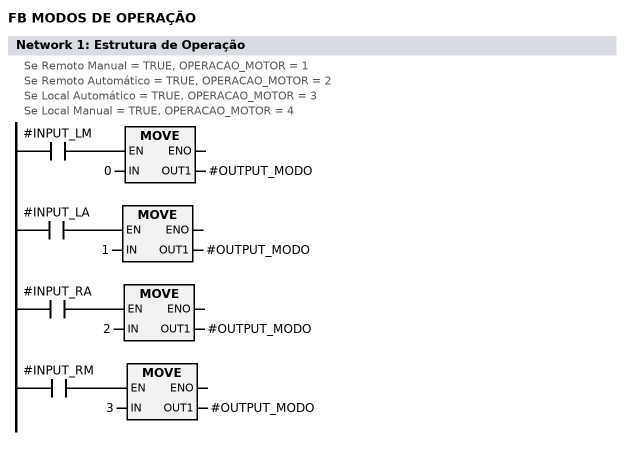
   RUNG wire#powerrail
      Contact( #INPUT_LM )
      Move(in := 0, out1 => #OUTPUT_MODO)
   END_RUNG
   RUNG wire#powerrail
      Contact( #INPUT_LA )
      Move(in := 1, out1 => #OUTPUT_MODO)
   END_RUNG
   RUNG wire#powerrail
      Contact( #INPUT_RA )
      Move(in := 2, out1 => #OUTPUT_MODO)
   END_RUNG
   RUNG wire#powerrail
      Contact( #INPUT_RM )
      Move(in := 3, out1 => #OUTPUT_MODO)
   END_RUNG
   // the same network as SCL:
   IF #INPUT_LM THEN #OUTPUT_MODO := 0; END_IF;
   IF #INPUT_LA THEN #OUTPUT_MODO := 1; END_IF;
   IF #INPUT_RA THEN #OUTPUT_MODO := 2; END_IF;
   IF #INPUT_RM THEN #OUTPUT_MODO := 3; END_IF;
END_REGION
END_FUNCTION_BLOCK

FUNCTION_BLOCK "FB_PARTIDA_INVERSOR"   // FB11, LAD
TITLE = Function Block PARTIDA INVERSOR
{ S7_Optimized_Access := 'TRUE' }
VERSION : 0.1
// Bloco para configurar os sinais de pulso (liga e desliga) em conjunto com 2 relés
   VAR_INPUT
      IN_LIGA_BOMBA : Bool;   // Entrada do comando para ligar a bomba
      IN_SUCÇÃO_OK : Bool;   // 0 = Sucção OK, permite ligar a bomba
      IN_OBSTRUÇÃO : Bool;   // 0 = Obstrução na pista
      IN_SOBRETORQUE : Bool;   // 0 = Sobretorque do motor/bomba
      IN_FALHA : Bool;   // 1 = Bomba em falha, comando desliga é pulsado
      IN_LIGADO : Bool;   // 1 = Bomba Ligada
      IN_HABILITA_CMB : Bool;   // Habilita bomba (Principal / Reserva)
      IN_LIGA_BOMBA_AUTO : Bool;
   END_VAR
   VAR_OUTPUT
      OUT_LIGA : Bool;   // Saída digital para ligar o Inversor
      OUT_DESLIGA : Bool;   // Saída digital para desligar o Inversor
   END_VAR
   VAR
      TEMP_LIGA : IEC_TIMER;   // Temporizador para simular o pulso de liga (0.5s)
      TEMP_DESLIGA : IEC_TIMER;   // Temporizador para simular o pulso de desliga (0.5s)
      DESLIGA_BOMBA : Bool;   // Memória auxiliar para desligar o Inversor
      OUT_TEST : Bool;
   END_VAR
BEGIN

REGION Network 1: Saída digital para ligar o Inversor
   // Condições para ligar:
   // IN_LIGA_BOMBA = 1, Sinal de liga recebido do bloco CONDIÇÃO DE PARTIDA
   // IN_SUCÇÃO = 1, Significa que a bomba está com sucção OK
   // IN_OBSTRUÇÃO = 0, Significa que não há obstrução na pista
   // IN_SOBRETORQUE = 0, Significa que não há alarme de sobretorque do motor/bomba
   // OUT_DESLIGA = 1, Para ligar, é necessário que a entrada digital de desliga no inversor (STOP) esteja com sinal alto, 
   // aguardando que o mesmo seja cortado com um pulso para desligar.
   // - Para desligar é necessário que o motor/bomba esteja enviando sinal de ligado.
   // 
   // Pulso para ligar: Configurado com um tempo de 0.5S
   // Pulso para desligar: Configurado com um tempo de 0.5S
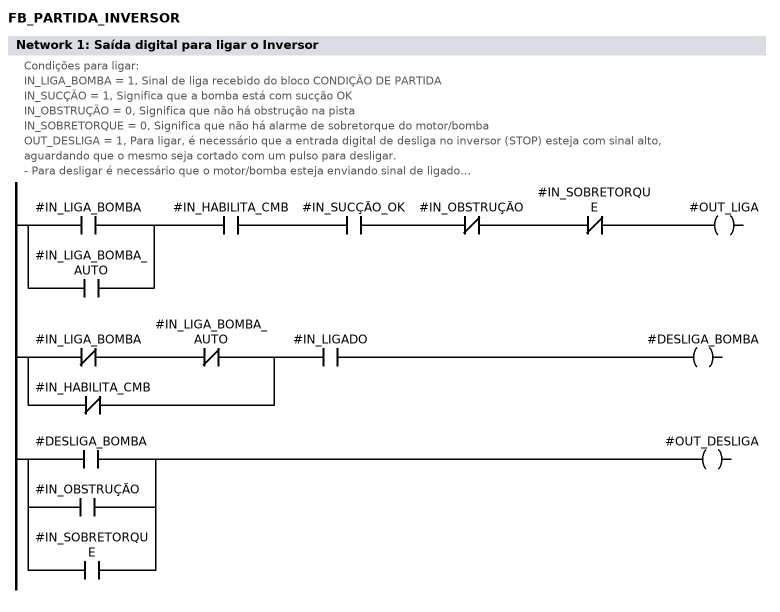
   RUNG wire#powerrail
      Contact( #IN_LIGA_BOMBA )
      wire#w1
      Contact( #IN_HABILITA_CMB )
      Contact( #IN_SUCÇÃO_OK )
      I_Contact( #IN_OBSTRUÇÃO )
      I_Contact( #IN_SOBRETORQUE )
      Coil( #OUT_LIGA )
   END_RUNG
   RUNG wire#powerrail
      Contact( #IN_LIGA_BOMBA_AUTO )
   END_RUNG wire#w1
   RUNG wire#powerrail
      I_Contact( #IN_LIGA_BOMBA )
      I_Contact( #IN_LIGA_BOMBA_AUTO )
      wire#w2
      Contact( #IN_LIGADO )
      Coil( #DESLIGA_BOMBA )
   END_RUNG
   RUNG wire#powerrail
      I_Contact( #IN_HABILITA_CMB )
   END_RUNG wire#w2
   RUNG wire#powerrail
      Contact( #DESLIGA_BOMBA )
      wire#w3
      Coil( #OUT_DESLIGA )
   END_RUNG
   RUNG wire#powerrail
      Contact( #IN_OBSTRUÇÃO )
   END_RUNG wire#w3
   RUNG wire#powerrail
      Contact( #IN_SOBRETORQUE )
   END_RUNG wire#w3
   // the same network as SCL:
   #OUT_LIGA := (#IN_LIGA_BOMBA OR #IN_LIGA_BOMBA_AUTO) AND #IN_HABILITA_CMB AND #IN_SUCÇÃO_OK AND NOT #IN_OBSTRUÇÃO AND NOT #IN_SOBRETORQUE;
   #DESLIGA_BOMBA := ((NOT #IN_LIGA_BOMBA AND NOT #IN_LIGA_BOMBA_AUTO) OR NOT #IN_HABILITA_CMB) AND #IN_LIGADO;
   #OUT_DESLIGA := #DESLIGA_BOMBA OR #IN_OBSTRUÇÃO OR #IN_SOBRETORQUE;
END_REGION
END_FUNCTION_BLOCK

FUNCTION_BLOCK "FB SUCÇÃO OK"   // FB15, LAD
TITLE = Function Block FB SUCÇÃO OK
{ S7_Optimized_Access := 'TRUE' }
VERSION : 0.1
   VAR_INPUT
      REFERENCIA : Real;   // Referência analógica em relação à sucção da bomba
      CADASTRO_SUCÇAO_INSUFICIENTE : Real;   // Cadastro de nível/pressão insuficiente
      CADASTRO_TEMPO_RESET : Time;   // Cadastro do tempo para resetar o alarme de Pressão Insuficiente
   END_VAR
   VAR_OUTPUT
      SUCÇÃO_OK : Bool;   // Sucção OK para operação
   END_VAR
   VAR
      SUCCAO_INSUFICIENTE : Bool;   // Sucção Insuficiente para operação
      RESET_ALARME : IEC_TIMER;   // Reset alarme de Sucção Insuficiente
   END_VAR
BEGIN

REGION Network 1: Set e Reset da Referência de Sucção insuficiente
   // Se nível for menor que a referência do Reservatório SUCÇÃO INSUFICIENTE,  bomba não pode ligar.
   // Caso o Nivel seja maior que a refêrencia então, após tempo cadastrado a bomba está habita para ligar
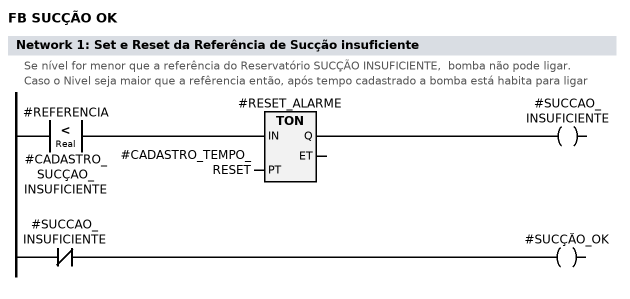
   #RESET_ALARME.TON(IN := #REFERENCIA < #CADASTRO_SUCÇAO_INSUFICIENTE, PT := #CADASTRO_TEMPO_RESET);
   #SUCCAO_INSUFICIENTE := #RESET_ALARME.Q;
   #SUCÇÃO_OK := NOT #SUCCAO_INSUFICIENTE;
END_REGION
END_FUNCTION_BLOCK

FUNCTION_BLOCK "FB VALVULA"   // FB17, LAD
{ S7_Optimized_Access := 'TRUE' }
VERSION : 0.1
// Network 1: Gerenciamento Status Válvula
// Network 2: Recebimento dos sinais de entrada (Sinais de campo e comandos)
// Network 3: MODO MANUAL: Conjunto de condições para ligar e desligar
// Network 4: MODO AUTOMÁTICO: Conjunto de condições para ligar e desligar
// Network 5: FALHA: Condicionamento de falha
// Network 6: LIGA BOMBA: Validando intertravamentos para ligar
// Network 7: ABRE VÁLVULA: Validando intertravamentos para abrir
   VAR_INPUT
      INPUT_ABERTA : Bool;   // 1 = Sinal elétrico de campo indicando válvula aberta
      INPUT_FECHADA : Bool;   // 1 = Sinal elétrico de campo indicando válvula fechada
      INPUT_FALHA : Bool;   // 0 = Sinal elétrico de campo indicando válvula em falha
      INPUT_LOCAL : Bool;   // 1 = Sinal elétrico de campo indicando válvula em modo local
      INPUT_REMOTO : Bool;   // 1 = Sinal elétrico de campo indicando válvula em modo remoto
      INPUT_FALHA_PROFINET : Bool;   // 1 = Indica falta de comunicação PROFINET com o equipamento
      INPUT_LIGA_AUTO : Bool;   // 1= indica que o processo pode ser ligado remoto manual
      PARAMETRO_ABRE : Bool;   // Parâmetro utilizado para abrir a válvula em modo automático
      PARAMETRO_FECHA : Bool;   // Parâmetro utilizado para fechar a válvula em modo automático
      CMD_ABRE : Bool;   // Comando enviado da IHM/SCADA para abrir a válvula
      CMD_MANUTEN : Bool;   // Comando enviado da IHM/SCADA para colocar a válvula em Modo de Manutenção
      CMD_MODO : Bool;   // Comando enviado da IHM/SCADA para colocar a bomba em (0 = Modo Manual, 1 = Modo Automático)
   END_VAR
   VAR_OUTPUT
      STATUS_VALV : Byte;   // 0 = FECHADA; 1 = ABERTA; 2 = FALHA
      ABRE_VALVULA : Bool;   // Saída acionada para abrir a válvula remotamente
      FECHA_VALVULA : Bool;   // Saída acionada para fechar a válvula remotamente
      REMOTO_MAN : Bool;   // Modo de Operação Remoto Manual
      REMOTO_AUTO : Bool;   // Modo de Operação Remoto Automático
      LOCAL_MAN : Bool;   // Modo de Operação Local Manual
   END_VAR
   VAR
      MANUTEN : Bool;   // Variável local para Indicar bomba em Modo Manutenção
      REMOTO : Bool;   // Variável local para indicar Modo Remoto
      FALHA : Bool;   // Variável local para Válvula em Falha
      ABRE_REM_MAN : Bool;   // Variável local para Acionamento Remoto Manual
      ABRE_REM_AUTO : Bool;   // Variável local para Acionamento Remoto Automático
   END_VAR
   VAR_TEMP   // added for the SCL form of the ladder/FBD networks
      _w1 : Bool;
   END_VAR
BEGIN

REGION Network 1: Gerenciamento Status Válvula
   // INPUT_ABERTA = Entrada de sinal de Válvula Aberta
   // INPUT_FECHADA = Entrada de sinal de Válvula Fechada
   // INPUT_FALHA = Entrada de sinal de Válvula em Falha
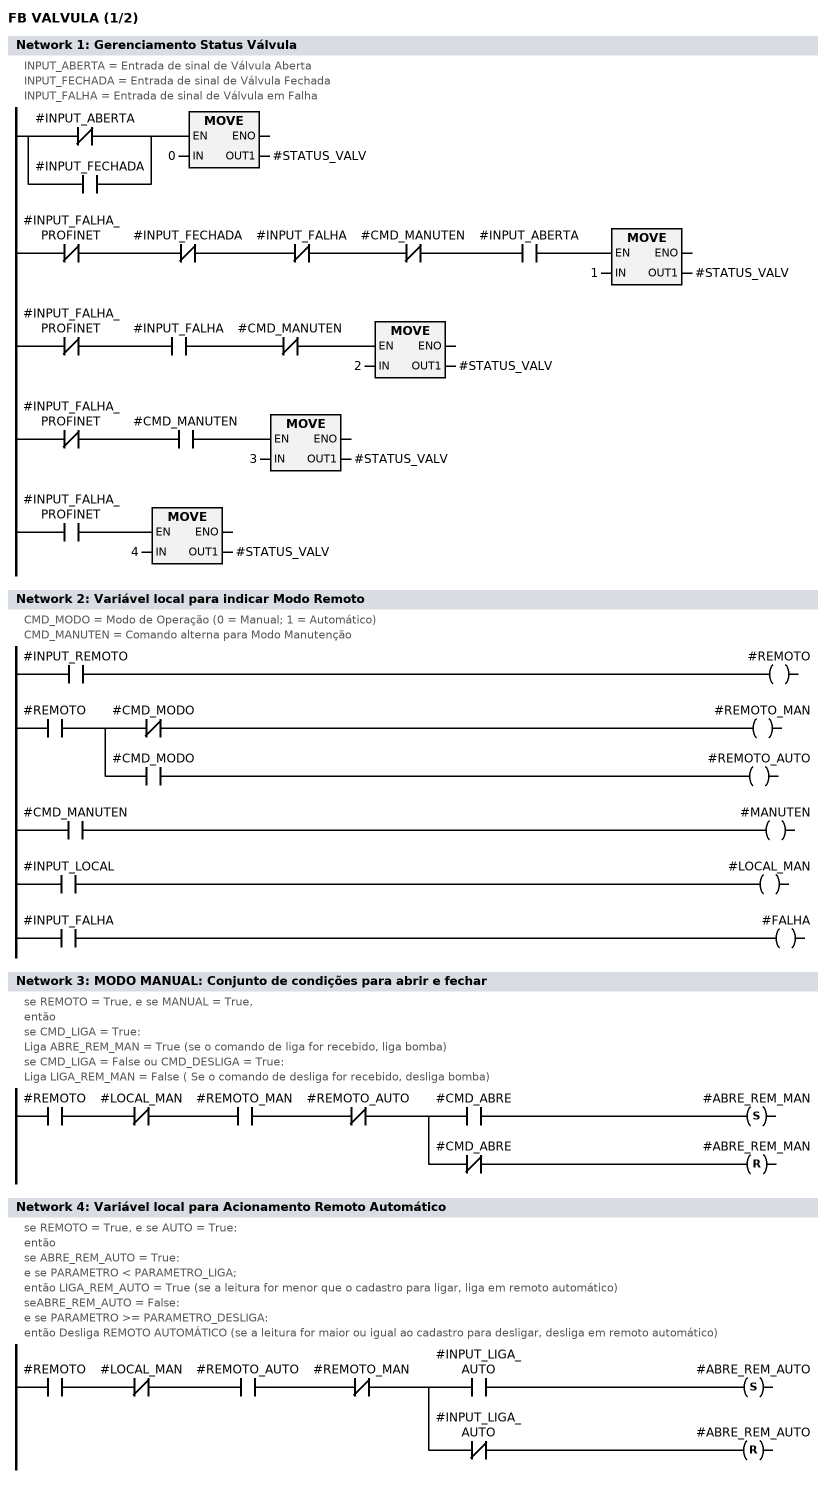
   RUNG wire#powerrail
      I_Contact( #INPUT_ABERTA )
      wire#w1
      Move(in := 0, out1 => #STATUS_VALV)
   END_RUNG
   RUNG wire#powerrail
      Contact( #INPUT_FECHADA )
   END_RUNG wire#w1
   RUNG wire#powerrail
      I_Contact( #INPUT_FALHA_PROFINET )
      I_Contact( #INPUT_FECHADA )
      I_Contact( #INPUT_FALHA )
      I_Contact( #CMD_MANUTEN )
      Contact( #INPUT_ABERTA )
      Move(in := 1, out1 => #STATUS_VALV)
   END_RUNG
   RUNG wire#powerrail
      I_Contact( #INPUT_FALHA_PROFINET )
      Contact( #INPUT_FALHA )
      I_Contact( #CMD_MANUTEN )
      Move(in := 2, out1 => #STATUS_VALV)
   END_RUNG
   RUNG wire#powerrail
      I_Contact( #INPUT_FALHA_PROFINET )
      Contact( #CMD_MANUTEN )
      Move(in := 3, out1 => #STATUS_VALV)
   END_RUNG
   RUNG wire#powerrail
      Contact( #INPUT_FALHA_PROFINET )
      Move(in := 4, out1 => #STATUS_VALV)
   END_RUNG
   // the same network as SCL:
   IF NOT #INPUT_ABERTA OR #INPUT_FECHADA THEN #STATUS_VALV := 0; END_IF;
   IF NOT #INPUT_FALHA_PROFINET AND NOT #INPUT_FECHADA AND NOT #INPUT_FALHA AND NOT #CMD_MANUTEN AND #INPUT_ABERTA THEN
       #STATUS_VALV := 1;
   END_IF;
   IF NOT #INPUT_FALHA_PROFINET AND #INPUT_FALHA AND NOT #CMD_MANUTEN THEN #STATUS_VALV := 2; END_IF;
   IF NOT #INPUT_FALHA_PROFINET AND #CMD_MANUTEN THEN #STATUS_VALV := 3; END_IF;
   IF #INPUT_FALHA_PROFINET THEN #STATUS_VALV := 4; END_IF;
END_REGION

REGION Network 2: Variável local para indicar Modo Remoto
   // CMD_MODO = Modo de Operação (0 = Manual; 1 = Automático)
   // CMD_MANUTEN = Comando alterna para Modo Manutenção
   RUNG wire#powerrail
      Contact( #INPUT_REMOTO )
      Coil( #REMOTO )
   END_RUNG
   RUNG wire#powerrail
      Contact( #REMOTO )
      wire#w1
      I_Contact( #CMD_MODO )
      Coil( #REMOTO_MAN )
   END_RUNG
   RUNG wire#w1
      Contact( #CMD_MODO )
      Coil( #REMOTO_AUTO )
   END_RUNG
   RUNG wire#powerrail
      Contact( #CMD_MANUTEN )
      Coil( #MANUTEN )
   END_RUNG
   RUNG wire#powerrail
      Contact( #INPUT_LOCAL )
      Coil( #LOCAL_MAN )
   END_RUNG
   RUNG wire#powerrail
      Contact( #INPUT_FALHA )
      Coil( #FALHA )
   END_RUNG
   // the same network as SCL:
   #REMOTO := #INPUT_REMOTO;
   #REMOTO_MAN := #REMOTO AND NOT #CMD_MODO;
   #REMOTO_AUTO := #REMOTO AND #CMD_MODO;
   #MANUTEN := #CMD_MANUTEN;
   #LOCAL_MAN := #INPUT_LOCAL;
   #FALHA := #INPUT_FALHA;
END_REGION

REGION Network 3: MODO MANUAL: Conjunto de condições para abrir e fechar
   // se REMOTO = True, e se MANUAL = True,
   // 
   // então
   // se CMD_LIGA = True: 
   // Liga ABRE_REM_MAN = True (se o comando de liga for recebido, liga bomba)
   // 
   // se CMD_LIGA = False ou CMD_DESLIGA = True:
   // Liga LIGA_REM_MAN = False ( Se o comando de desliga for recebido, desliga bomba)
   RUNG wire#powerrail
      Contact( #REMOTO )
      I_Contact( #LOCAL_MAN )
      Contact( #REMOTO_MAN )
      I_Contact( #REMOTO_AUTO )
      wire#w1
      Contact( #CMD_ABRE )
      S_Coil( #ABRE_REM_MAN )
   END_RUNG
   RUNG wire#w1
      I_Contact( #CMD_ABRE )
      R_Coil( #ABRE_REM_MAN )
   END_RUNG
   // the same network as SCL:
   #_w1 := #REMOTO AND NOT #LOCAL_MAN AND #REMOTO_MAN AND NOT #REMOTO_AUTO;
   IF #_w1 AND #CMD_ABRE THEN #ABRE_REM_MAN := TRUE; END_IF;
   IF #_w1 AND NOT #CMD_ABRE THEN #ABRE_REM_MAN := FALSE; END_IF;
END_REGION

REGION Network 4: Variável local para Acionamento Remoto Automático
   // se REMOTO = True, e se AUTO = True:
   // 
   // então
   // se ABRE_REM_AUTO = True:
   // e se PARAMETRO < PARAMETRO_LIGA;
   // então LIGA_REM_AUTO = True (se a leitura for menor que o cadastro para ligar, liga em remoto automático)
   // 
   // seABRE_REM_AUTO = False:
   // e se PARAMETRO >= PARAMETRO_DESLIGA:
   // então Desliga REMOTO AUTOMÁTICO (se a leitura for maior ou igual ao cadastro para desligar, desliga em remoto automático)
   RUNG wire#powerrail
      Contact( #REMOTO )
      I_Contact( #LOCAL_MAN )
      Contact( #REMOTO_AUTO )
      I_Contact( #REMOTO_MAN )
      wire#w1
      Contact( #INPUT_LIGA_AUTO )
      S_Coil( #ABRE_REM_AUTO )
   END_RUNG
   RUNG wire#w1
      I_Contact( #INPUT_LIGA_AUTO )
      R_Coil( #ABRE_REM_AUTO )
   END_RUNG
   // the same network as SCL:
   #_w1 := #REMOTO AND NOT #LOCAL_MAN AND #REMOTO_AUTO AND NOT #REMOTO_MAN;
   IF #_w1 AND #INPUT_LIGA_AUTO THEN #ABRE_REM_AUTO := TRUE; END_IF;
   IF #_w1 AND NOT #INPUT_LIGA_AUTO THEN #ABRE_REM_AUTO := FALSE; END_IF;
END_REGION

REGION Network 5: FALHA: Condicionamento de falha
   // se FALHA = False;
   // 
   // então
   // ABRE_REM_AUTO = False (Reseta Liga Remoto Automático)
   // ABRE_REM_MAN = False (Reseta Liga Remoto Manual)
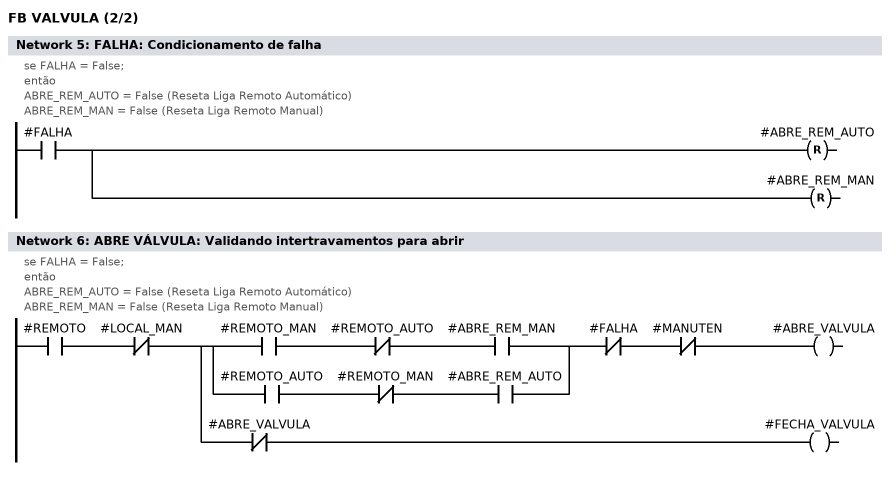
   RUNG wire#powerrail
      Contact( #FALHA )
      wire#w1
      R_Coil( #ABRE_REM_AUTO )
   END_RUNG
   RUNG wire#w1
      R_Coil( #ABRE_REM_MAN )
   END_RUNG
   // the same network as SCL:
   IF #FALHA THEN
       #ABRE_REM_AUTO := FALSE;
       #ABRE_REM_MAN := FALSE;
   END_IF;
END_REGION

REGION Network 6: ABRE VÁLVULA: Validando intertravamentos para abrir
   // se FALHA = False;
   // 
   // então
   // ABRE_REM_AUTO = False (Reseta Liga Remoto Automático)
   // ABRE_REM_MAN = False (Reseta Liga Remoto Manual)
   RUNG wire#powerrail
      Contact( #REMOTO )
      I_Contact( #LOCAL_MAN )
      wire#w1
      Contact( #REMOTO_MAN )
      I_Contact( #REMOTO_AUTO )
      Contact( #ABRE_REM_MAN )
      wire#w2
      I_Contact( #FALHA )
      I_Contact( #MANUTEN )
      Coil( #ABRE_VALVULA )
   END_RUNG
   RUNG wire#w1
      Contact( #REMOTO_AUTO )
      I_Contact( #REMOTO_MAN )
      Contact( #ABRE_REM_AUTO )
   END_RUNG wire#w2
   RUNG wire#w1
      I_Contact( #ABRE_VALVULA )
      Coil( #FECHA_VALVULA )
   END_RUNG
   // the same network as SCL:
   #_w1 := #REMOTO AND NOT #LOCAL_MAN;
   #ABRE_VALVULA := #_w1 AND ((#REMOTO_MAN AND NOT #REMOTO_AUTO AND #ABRE_REM_MAN) OR (#REMOTO_AUTO AND NOT #REMOTO_MAN AND #ABRE_REM_AUTO)) AND NOT #FALHA AND NOT #MANUTEN;
   #FECHA_VALVULA := #_w1 AND NOT #ABRE_VALVULA;
END_REGION
END_FUNCTION_BLOCK

FUNCTION_BLOCK "FB INTERTRAVAMENTO_PAINEL"   // FB27, SCL
{ S7_Optimized_Access := 'TRUE' }
VERSION : 0.1
   VAR_INPUT
      INPUT_BT_EMERGENCIA : Bool;
      INPUT_DISJUNTOR : Bool;
      INPUT_FONTE1 : Bool;
      INPUT_FONTE2 : Bool;
      INPUT_RELE_FALTA : Bool;
      INPUT_CONDICAO : Bool;
      INPUT_TESTE : Bool;
   END_VAR
   VAR_OUTPUT
      OUTPUT_PAINEL_OK : Bool;
   END_VAR
BEGIN

   IF ((#INPUT_BT_EMERGENCIA AND // Supondo que BT_EMERGENCIA é True quando ñ ATUADO
         NOT #INPUT_DISJUNTOR AND
         #INPUT_FONTE1 AND
         #INPUT_FONTE2 AND
         #INPUT_RELE_FALTA AND // Supondo que RELE_FALTA é True quando ñ ATUADO
         #INPUT_CONDICAO) 
      OR
      #INPUT_TESTE) THEN // teste força a saída 
   #OUTPUT_PAINEL_OK := TRUE;
   ELSE
       #OUTPUT_PAINEL_OK := FALSE;
   END_IF;
END_FUNCTION_BLOCK

// folder: 1. FB Bilbiotecas/1.1 Acionamento/1.1.1 Inversores

FUNCTION_BLOCK "FB AFERIÇÃO INVERSORES"   // FB2, LAD
{ S7_Optimized_Access := 'TRUE' }
VERSION : 0.1
// Os sinais de campo são recebidos em corrente (4-20mA) e representados pelo fundo de escala do CLP. Este bloco faz a conversão do sinal para a leitura real da medição.
// 
// Network 1: Ajuste do fundo de escala aos parâmetros de aferição
// Network 2: Cálculo da equação da reta para definir a leitura atual da entrada analógica
// Network 3: Setando o alarme SEM 4mA na entrada digital caso seja rompida
   VAR_INPUT
      ANALOG_IN_4a20mA : Int;   // Entrada do sinal analógico
      Y1_CONFIG : Int;   // Fundo de escala mínimo para o CLP
      Y2_CONFIG : Int;   // Fundo de escala máximo para o CLP
      X1_CONFIG : Int;   // Fundo de escala mínimo para o equipamento
      X2_CONFIG : Int;   // Fundo de escala máximo para o equipamento
      COMANDO : Int;   // Comando enviado da IHM/SCADA para aferir determinado equipamento
      COMANDO_VALOR : Int;   // Valor comparativo para executar o Bloco FB
      GRANDEZA_MAX : Int;   // Referência a grandeza maxima no qual o bloco vai utilizar para fazer a curva da reta
   END_VAR
   VAR_OUTPUT
      ANALOG_OUT_4a20mA : Real;   // Saída do sinal analógico já aferido
      ALARME_SEM_4mA : Bool;   // 1 = Entrada sem 4mA, indicando erro; 0 = Entrada OK
      RANGE_MIN_CADASTRADO : Int;   // Valor do cadastro máximo armazenado para visualizar na IHM
      RANGE_MAX_CADASTRADO : Int;   // Valor do cadastro mínimo armazenado para visualizar na IHM
   END_VAR
   VAR
      ANALOG_IN_LIMITED : Int;   // Tratamento de erro do sinal analógico para capturar apenas leituras que estão dentro do range do CLP
      ANALOG_IN_LIMITED_REAL : UInt;   // Saída do sinal ajustado conforme a grandeza máxima
      STATIC_X1 : UInt;   // Fundo de escala mínimo para o equipamento (Instanciado no FB)
      STATIC_X2 : UInt;   // Fundo de escala máximo para o equipamento (Instanciado no FB)
      STATIC_Y1 : UInt;   // Fundo de escala mínimo para o CLP (Instanciado no FB)
      STATIC_Y2 : UInt;   // Fundo de escala máximo para o CLP (Instanciado no FB)
      STATIC_GRANDEZA_MAX : UInt;   // Grandeza máxima do equipamento
      AJUSTAR_CURVA : Bool;   // Memória para mover as entradas às instâncias
      PONTO_ZERO : Int;   // Range mínimo do equipamento quando é diferente de 0
      ALARME_RESET : TOF_TIME;   // Reset do alarme Sem 4mA ao estabilizar o sinal
      PULSO_AJUSTAR : Bool;   // Pulso para realizar a aferição da curva
   END_VAR
   VAR_TEMP   // added for the SCL form of the ladder/FBD networks
      _w1 : Bool;
   END_VAR
BEGIN

REGION Network 1: Ajuste do fundo de escala aos parâmetros de aferição
   // X1_CONFIG = Fundo de escala mínimo para o equipamento
   // X2_CONFIG = Fundo de escala máximo para o equipamento
   // Y1_CONFIG = Fundo de escala mínimo para o CLP
   // Y2_CONFIG = Fundo de escala máximo para o CLP
   // GRANDEZA_MAX = Referência a grandeza maxima no qual o bloco vai utilizar para fazer a curva da reta
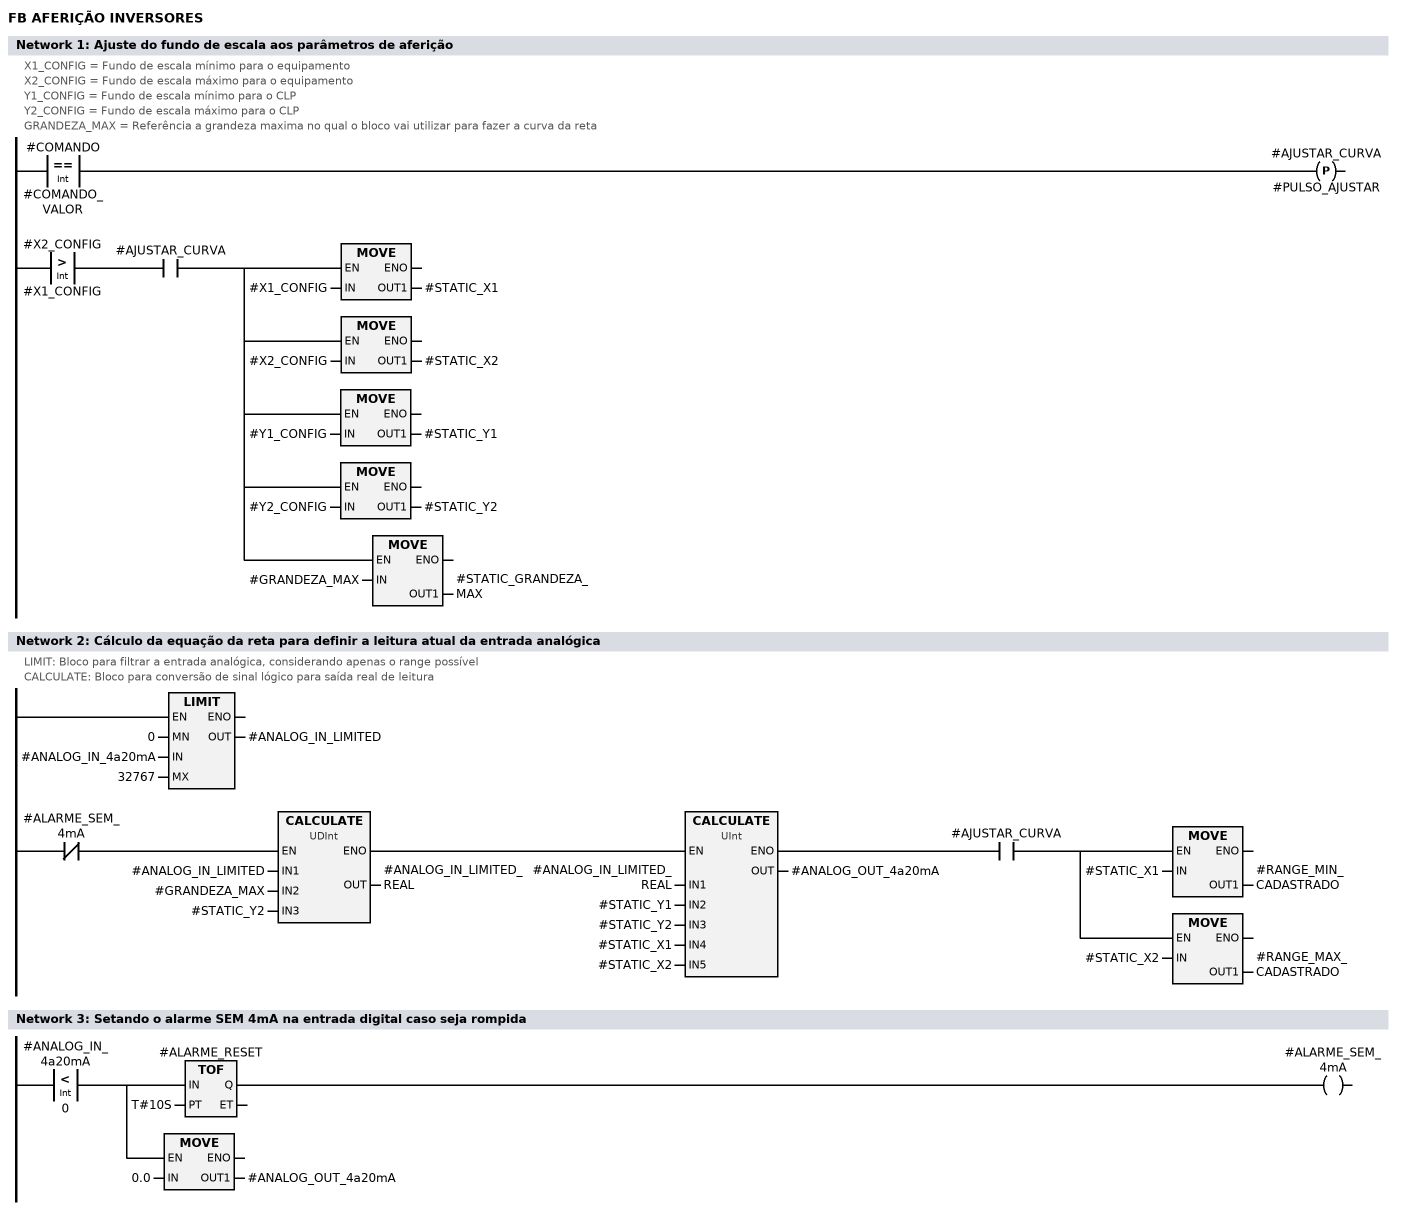
   #_w1 := #COMANDO = #COMANDO_VALOR;
   #AJUSTAR_CURVA := #_w1 AND NOT #PULSO_AJUSTAR;   // rising edge
   #PULSO_AJUSTAR := #_w1;
   IF (#X2_CONFIG > #X1_CONFIG) AND #AJUSTAR_CURVA THEN
       #STATIC_X1 := #X1_CONFIG;
       #STATIC_X2 := #X2_CONFIG;
       #STATIC_Y1 := #Y1_CONFIG;
       #STATIC_Y2 := #Y2_CONFIG;
       #STATIC_GRANDEZA_MAX := #GRANDEZA_MAX;
   END_IF;
END_REGION

REGION Network 2: Cálculo da equação da reta para definir a leitura atual da entrada analógica
   // LIMIT: Bloco para filtrar a entrada analógica, considerando apenas o range possível
   // CALCULATE: Bloco para conversão de sinal lógico para saída real de leitura
   #ANALOG_IN_LIMITED := LIMIT(MN := 0, IN := #ANALOG_IN_4a20mA, MX := 32767);
   IF NOT #ALARME_SEM_4mA THEN
       #ANALOG_IN_LIMITED_REAL := #ANALOG_IN_LIMITED * #STATIC_Y2 / #GRANDEZA_MAX;
       #ANALOG_OUT_4a20mA := (#ANALOG_IN_LIMITED_REAL - #STATIC_Y1) * (#STATIC_X2 - #STATIC_X1) / (#STATIC_Y2 - #STATIC_Y1);
   END_IF;
   IF NOT #ALARME_SEM_4mA AND #AJUSTAR_CURVA THEN
       #RANGE_MIN_CADASTRADO := #STATIC_X1;
       #RANGE_MAX_CADASTRADO := #STATIC_X2;
   END_IF;
END_REGION

REGION Network 3: Setando o alarme SEM 4mA na entrada digital caso seja rompida
   #_w1 := #ANALOG_IN_4a20mA < 0;
   #ALARME_RESET(IN := #_w1, PT := T#10S);   // TOF
   #ALARME_SEM_4mA := #ALARME_RESET.Q;
   IF #_w1 THEN #ANALOG_OUT_4a20mA := 0.0; END_IF;
END_REGION
END_FUNCTION_BLOCK

FUNCTION_BLOCK "FB STATUS ECSX"   // FB12, LAD
TITLE = Function Block STATUS ECSX - Status dos exaustores (ECS1 - ECS2 - ECS3)
{ S7_Optimized_Access := 'TRUE' }
VERSION : 0.1
// Sinais de status (ligado e falha) recebidos de campo
   VAR_INPUT
      INPUT_LIGADO : Bool;   // Entrada do sinal de Motor/Bomba ligado
      INPUT_FALHA : Bool;   // Entrada do sinal de falha instanciado na Network 1
      INPUT_MANUTEN : Bool;   // Entrada do sinal de manutenção instanciado na Network 1
      INPUT_FALHA_PROFINET : Bool;   // 1 = Indica falta de comunicação PROFINET com o equipamento
   END_VAR
   VAR_OUTPUT
      STATUS_MOTOR : Byte;   // Indicador de Status do exaustor
   END_VAR
BEGIN

REGION Network 1: Acionamento do status ligado
   // INUPT_LIGADO = TRUE: Exaustor ligado
   // INPUT_FALHA = TRUE: Exaustor em falha
   // INPUT_FALHA_PROFINET = TRUE: Sem Comunicação PROFINET
   // INPUT_MANUTEN = TRUE: Motor/Exaustor em manutenção
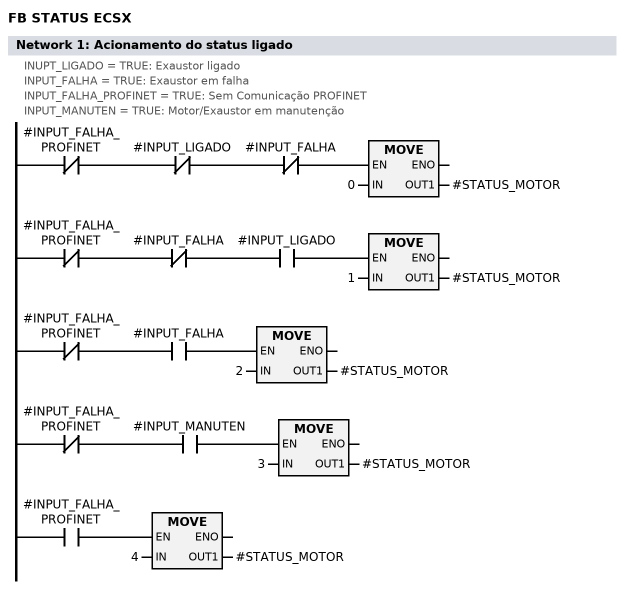
   RUNG wire#powerrail
      I_Contact( #INPUT_FALHA_PROFINET )
      I_Contact( #INPUT_LIGADO )
      I_Contact( #INPUT_FALHA )
      Move(in := 0, out1 => #STATUS_MOTOR)
   END_RUNG
   RUNG wire#powerrail
      I_Contact( #INPUT_FALHA_PROFINET )
      I_Contact( #INPUT_FALHA )
      Contact( #INPUT_LIGADO )
      Move(in := 1, out1 => #STATUS_MOTOR)
   END_RUNG
   RUNG wire#powerrail
      I_Contact( #INPUT_FALHA_PROFINET )
      Contact( #INPUT_FALHA )
      Move(in := 2, out1 => #STATUS_MOTOR)
   END_RUNG
   RUNG wire#powerrail
      I_Contact( #INPUT_FALHA_PROFINET )
      Contact( #INPUT_MANUTEN )
      Move(in := 3, out1 => #STATUS_MOTOR)
   END_RUNG
   RUNG wire#powerrail
      Contact( #INPUT_FALHA_PROFINET )
      Move(in := 4, out1 => #STATUS_MOTOR)
   END_RUNG
   // the same network as SCL:
   IF NOT #INPUT_FALHA_PROFINET AND NOT #INPUT_LIGADO AND NOT #INPUT_FALHA THEN #STATUS_MOTOR := 0; END_IF;
   IF NOT #INPUT_FALHA_PROFINET AND NOT #INPUT_FALHA AND #INPUT_LIGADO THEN #STATUS_MOTOR := 1; END_IF;
   IF NOT #INPUT_FALHA_PROFINET AND #INPUT_FALHA THEN #STATUS_MOTOR := 2; END_IF;
   IF NOT #INPUT_FALHA_PROFINET AND #INPUT_MANUTEN THEN #STATUS_MOTOR := 3; END_IF;
   IF #INPUT_FALHA_PROFINET THEN #STATUS_MOTOR := 4; END_IF;
END_REGION
END_FUNCTION_BLOCK

FUNCTION_BLOCK "FB INVERSOR SIEMENS"   // FB20, LAD
{ S7_Optimized_Access := 'TRUE' }
VERSION : 0.1
   VAR_INPUT
      RPM_min_Driver : Int;
      RPM_Max_Driver : Int;
      Setpoint_Velocidade : Int;
   END_VAR
   VAR_OUTPUT
      Telegram_Out_Velocidade : Int;
   END_VAR
   VAR_TEMP
      Aux_Velocidade : Real;
   END_VAR
BEGIN

REGION Network 1: Controle Velocidade
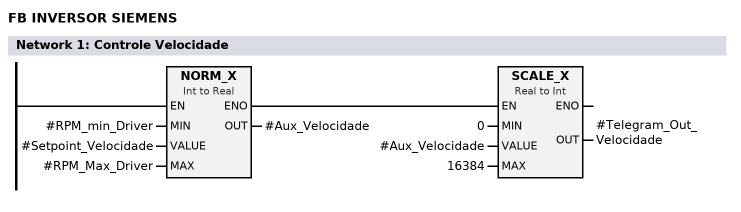
   RUNG wire#powerrail
      { S7_Templates := "[SrcType := Int, DestType := Real]" } Normalize(min := #RPM_min_Driver, value := #Setpoint_Velocidade, max := #RPM_Max_Driver, out => #Aux_Velocidade)
      { S7_Templates := "[SrcType := Real, DestType := Int]" } Scale(min := 0, value := #Aux_Velocidade, max := 16384, out => #Telegram_Out_Velocidade)
   END_RUNG
   // the same network as SCL:
   #Aux_Velocidade := NORM_X(MIN := #RPM_min_Driver, VALUE := #Setpoint_Velocidade, MAX := #RPM_Max_Driver);
   #Telegram_Out_Velocidade := SCALE_X(MIN := 0, VALUE := #Aux_Velocidade, MAX := 16384);
END_REGION
END_FUNCTION_BLOCK

FUNCTION_BLOCK "SINA_SPEED_TLG20"   // FB38003, SCL
TITLE = Speed control S7 to SINAMICS using Standardtelegram 20
{ S7_Optimized_Access := 'TRUE' }
AUTHOR : SIEMENS
FAMILY : DRIVES
NAME : SINA_SPD_TLG20
VERSION : 1.0
// The function block SINA_SPEED_TLG20 controls a SINAMICS drive using standard telegram 20
   VAR_INPUT
      enableAxis : Bool;   // 0 -> 1 = Enable the drive (OFF2 / OFF 3 are 1 in default status) (OFF1 = 0->1)
      ackError : Bool;   // 0 -> 1 = Acknowledge drive error
      speedSp : Real;   // Speed setpoint [rpm]
      selectCDS : USInt;   // Selection of the Command Data Set (0 = CDS0, 1 = CDS1)
      refSpeed : Real;   // Reference speed [p2000] in [rpm]
      refCurrent : Real;   // Reference current [p2002] in [Aeff]
      refTorque : Real;   // Reference torque [p2003] in [Nm]
      refPower : Real;   // Reference power [r2005] in [kW]
      configAxis : Word := 16#003F;   // binary programmed input to control all functions in the telegram without its own function block input
      HWIDSTW : HW_IO;   // Hardware Identifer set point slot
      HWIDZSW : HW_IO;   // Hardware Identifer actual value slot
   END_VAR
   VAR_OUTPUT
      axisEnabled : Bool;   // 1 = Drive is enabled
      lockout : Bool;   // 1 = Drive lockout active
      actCDS : USInt;   // Active Command Data Set (0 = CDS0, 1 = CDS1)
      actSpeed : Real;   // Smoothed actual speed in [1/min]
      actCurrent : Real;   // Smoothed current actual in [Arms]
      actTorque : Real;   // Actual smoothed torque in [Nm]
      actPower : Real;   // Actual smoothed active power in [kW]
      faultVIKNAMUR : Word;   // Fault word according to the VIK-NAMUR defintion
      error : Bool;   // 1 = Error (FB and Infeed)
      status : Int;   // Status output (7002 = FB in operation; 7xxx = warning; 8xxx = error description - read the manual)
      diagId : Int;   // Error codes of the system function blocks DPWR / DPRD_DAT
   END_VAR
   VAR_TEMP
      tempSpeed : Real;   // Speed setpoint in percent
      tempRefValueInvalid : Bool;   // At least one reference value is 0 or < 0
      tempSendBuf : Array[0..1] of Word;   // Send buffer
      tempRecvBuf : Array[0..5] of Word;   // Receive buffer
   END_VAR
   VAR CONSTANT
      NORMALIZATION_VALUE : Int := 16#4000;   // Used to calculate the Real values
      MAX_INT : Int := 16#7FFF;
      MIN_INT : Int := 16#8000;
      REF_CURRRENT_INVALID : Int := 16#7010;   // RefCurrent input is 0 or < 0
      REF_TORQUE_INVALID : Int := 16#7011;   // RefTorque input is 0 or < 0
      REF_POWER_INVALID : Int := 16#7012;   // RefPower input is 0 or < 0
      REF_VALUES_INVALID : Int := 16#7013;   // Multiple reference values are 0 or < 0
      NO_ERROR : Int := 16#7002;   // No error
      ERROR_REF_SPEED_INVALID : Int := 16#8001;   // RefSpeed input is 0 or < 0
      ERROR_INVALID_CDS : Int := 16#8002;   // Invalid Command Data Set selected
      ERROR_DRIVE : Int := 16#8401;   // Drive error
      ERROR_LOCKOUT : Int := 16#8402;   // Drive lockout
      ERROR_DPREAD : Int := 16#8600;   // DPRD_DAT returned an error
      ERROR_DPWRITE : Int := 16#8601;   // DPWR_DAT returned an error
      ERROR_FAULT_WORD : Int := 16#8700;   // faultVIKNAMUR is not 0
      STW1 : USInt := 0;
      ZSW1 : USInt := 0;
      NSOLL_A : USInt := 1;
   END_VAR
BEGIN
   //=============================================================================
   //SIEMENS AG
   //(c)Copyright 2019 All Rights Reserved
   //-----------------------------------------------------------------------------
   // Library:       LSINAExt
   // Tested with:   SIMATIC S7 CPU 1513-1 PN V2.5
   // Engineering:   TIA Portal V15
   // Restrictions:  -
   // Requirements:  S7-1200 / S7-1500
   // Functionality: cyclic communication between a SINAMICS a PLC.
   //                If in HWConfig standard telegram 20 are projected 2 PZD-words are exchanged
   //                in every bus cycle.
   //                The parametrisation of these words is described in the manual of the
   //                SINAMICS
   //-----------------------------------------------------------------------------
   //Change log table:
   //Version  Date       Expert in charge Changes applied
   //01.00.00 11.02.2019 (AS) First released version
   //=============================================================================

   // Prepare PZD1 (STW1)
   #tempSendBuf[#STW1].%X0 := #enableAxis;
   #tempSendBuf[#STW1].%X7 := #ackError;
   #tempSendBuf[#STW1].%X1 := #configAxis.%X0;
   #tempSendBuf[#STW1].%X2 := #configAxis.%X1;
   #tempSendBuf[#STW1].%X3 := #configAxis.%X2;
   #tempSendBuf[#STW1].%X4 := #configAxis.%X3;
   #tempSendBuf[#STW1].%X5 := #configAxis.%X4;
   #tempSendBuf[#STW1].%X6 := #configAxis.%X5;
   #tempSendBuf[#STW1].%X11 := #configAxis.%X6;
   #tempSendBuf[#STW1].%X15 := #selectCDS = 1; // true = CDS0, false = CDS1
   #tempSendBuf[#STW1].%X10 := TRUE; // control by PLC
   #tempSendBuf[#STW1].%X13 := FALSE; // STW1.X13 not used in Telegram 20
   #tempSendBuf[#STW1].%X14 := FALSE; // STW1.X14 not used in Telegram 20

   // Check CDS index
   IF (#selectCDS < 0)
       OR (#selectCDS > 1)
   THEN
       #error := TRUE;
       #status := #ERROR_INVALID_CDS;
       #tempSendBuf[#STW1].%X0 := FALSE; // disable axis
   END_IF;

   // Speed
   IF #refSpeed > 0 THEN
       #tempSpeed := #speedSp * (#NORMALIZATION_VALUE / #refSpeed);
       // Limit REAL - Variable to INT - limits
       IF #tempSpeed > #MAX_INT
       THEN
           #tempSpeed := #MAX_INT;
       ELSIF #tempSpeed < #MIN_INT
       THEN
           #tempSpeed := #MIN_INT;
       ELSE
           ; // not needed
       END_IF;
       #tempSendBuf[#NSOLL_A] := INT_TO_WORD(REAL_TO_INT(#tempSpeed));
   ELSE
       #error := TRUE;
       #status := #ERROR_REF_SPEED_INVALID;
       #tempSendBuf[#NSOLL_A] := W#16#0;
   END_IF;

   // Send telegram to drive
   #diagId := DPWR_DAT(LADDR := #HWIDSTW,
                       RECORD := #tempSendBuf);

   // Error when writing the telegram
   IF #diagId <> 0 THEN
       #error := TRUE;
       #status := #ERROR_DPWRITE;

       // Reset outputs
       #actSpeed := 0.0;
       #actCurrent := 0.0;
       #actTorque := 0.0;
       #actPower := 0.0;
       #faultVIKNAMUR := W#16#0;

       RETURN;
   ELSE
       ;
   END_IF;

   // Receive telegram from drive
   #diagId := DPRD_DAT(LADDR := #HWIDZSW,
                       RECORD => #tempRecvBuf);

   // Error when reading the telegram
   IF #diagId <> 0 THEN
       #error := TRUE;
       #status := #ERROR_DPREAD;

       // Reset outputs
       #actSpeed := 0.0;
       #actCurrent := 0.0;
       #actTorque := 0.0;
       #actPower := 0.0;
       #faultVIKNAMUR := W#16#0;

       RETURN;
   ELSE
       ;
   END_IF;

   // Analyse ZSW1
   #axisEnabled := #tempRecvBuf[#ZSW1].%X2;
   #lockout := #tempRecvBuf[#ZSW1].%X6;
   #error := #tempRecvBuf[#ZSW1].%X3 OR #tempRecvBuf[#ZSW1].%X6;

   IF #tempRecvBuf[#ZSW1].%X3 THEN
       #status := #ERROR_DRIVE;
   ELSIF #tempRecvBuf[#ZSW1].%X6 THEN
       #status := #ERROR_LOCKOUT;
   ELSE
       #status := #NO_ERROR;
   END_IF;

   // Check CDS
   IF #tempRecvBuf[#ZSW1].%X15 THEN
       #actCDS := 1;
   ELSE
       #actCDS := 0;
   END_IF;

   //IF #actCDS <> #selectCDS THEN
   //  #error := TRUE;
   //  #status := #ERROR_INVALID_CDS;
   //END_IF;

   // Actual speed
   IF (#refSpeed <= 0)
       AND #enableAxis
   THEN
       #actSpeed := 0.0;
       #error := TRUE;
       #status := #ERROR_REF_SPEED_INVALID;
   ELSE
       #actSpeed := INT_TO_REAL(WORD_TO_INT(#tempRecvBuf[1])) / (#NORMALIZATION_VALUE / #refSpeed);
   END_IF;

   // Actual current
   IF (#refCurrent <= 0)
       AND #enableAxis
       AND NOT #error
   THEN
       #actCurrent := 0.0;

       IF #tempRefValueInvalid THEN
           #status := #REF_VALUES_INVALID;
       ELSE
           #status := #REF_CURRRENT_INVALID;
           #tempRefValueInvalid := TRUE;
       END_IF;
   ELSE
       #actCurrent := INT_TO_REAL(WORD_TO_INT(#tempRecvBuf[2])) / (#NORMALIZATION_VALUE / #refCurrent);
   END_IF;

   // Actual torque
   IF (#refTorque <= 0)
       AND #enableAxis
       AND NOT #error
   THEN
       #actTorque := 0.0;

       IF #tempRefValueInvalid THEN
           #status := #REF_VALUES_INVALID;
       ELSE
           #status := #REF_TORQUE_INVALID;
           #tempRefValueInvalid := TRUE;
       END_IF;
   ELSE
       #actTorque := INT_TO_REAL(WORD_TO_INT(#tempRecvBuf[3])) / (#NORMALIZATION_VALUE / #refTorque);
   END_IF;

   // Actual active power
   IF (#refPower <= 0)
       AND #enableAxis
       AND NOT #error
   THEN
       #actPower := 0.0;

       IF #tempRefValueInvalid THEN
           #status := #REF_VALUES_INVALID;
       ELSE
           #status := #REF_POWER_INVALID;
           #tempRefValueInvalid := TRUE;
       END_IF;
   ELSE
       #actPower := INT_TO_REAL(WORD_TO_INT(#tempRecvBuf[4])) / (#NORMALIZATION_VALUE / #refPower);
   END_IF;

   // VIKNAMUR fault word
   #faultVIKNAMUR := #tempRecvBuf[5];
   IF #faultVIKNAMUR <> 16#0000 THEN
       #error := TRUE;
       #status := #ERROR_FAULT_WORD;
   ELSE
       ;
   END_IF;
END_FUNCTION_BLOCK

// ===== library: MasterCopy "FB CONTADOR" =====

// folder: 1. FB Bilbiotecas

FUNCTION_BLOCK "FB CONTADOR"   // FB7, LAD
TITLE = Function Block MINUTEIRO - Contador de Minutos
{ S7_Optimized_Access := 'TRUE' }
VERSION : 0.1
// Bloco para realizar a contagem de quantos minutos cada motor/bomba passou ligado.
   VAR_INPUT
      INPUT_LIGADO : Bool;   // Entrada do sinal de falha instanciado na Network 1
      INPUT_RESET_MINUTEIRO : Bool;   // Entrada do sinal de reset minuteiro (minutos trabalhadas da bomba)
   END_VAR
   VAR_OUTPUT
      SEGUNDEIRO : UInt;   // Saída do segundeiro (segundos trabalhados da bomba)
      MINUTEIRO : Real;   // Saída do minuteiro (minutos trabalhados da bomba)
      HORIMETRO : Real;   // Saída do horimetro (horas trabalhados da bomba)
   END_VAR
   VAR
      RESET_SEGUNDO : Bool;   // Comando para zerar os minutos acumuladas
      MINUTO : Bool;   // Pulso para contador de minutos
      COUNT_MINUTO : Bool;   // Contador de minutos
      RESET_MINUTO : Bool;   // Reset do contador de minutos
      SEGUNDOS : UInt;   // Segundos armazenados
      TIMER_SEGUNDO : IEC_COUNTER;   // Bloco contador de segundos
   END_VAR
BEGIN

REGION Network 1: Comando para zerar os minutos acumuladas
   // TIMER_SEGUNDO: Bloco contador de segundos
   // TIMER_MINUTO: Bloco contador de minutos
   // INC: Incremento de horas
   // RESET_MINUTEIRO: Comando para zerar os minutos acumulados
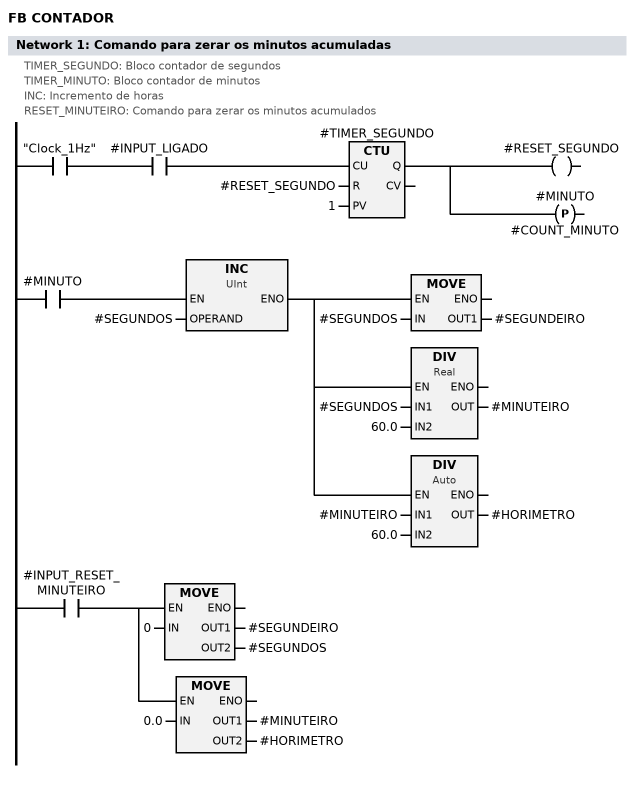
   #TIMER_SEGUNDO.CTU(CU := "Clock_1Hz" AND #INPUT_LIGADO, R := #RESET_SEGUNDO, PV := 1);
   #RESET_SEGUNDO := #TIMER_SEGUNDO.Q;
   #MINUTO := #TIMER_SEGUNDO.Q AND NOT #COUNT_MINUTO;   // rising edge
   #COUNT_MINUTO := #TIMER_SEGUNDO.Q;
   IF #MINUTO THEN
       #SEGUNDOS := #SEGUNDOS + 1;
       #SEGUNDEIRO := #SEGUNDOS;
       #MINUTEIRO := #SEGUNDOS / 60.0;
       #HORIMETRO := #MINUTEIRO / 60.0;
   END_IF;
   IF #INPUT_RESET_MINUTEIRO THEN
       #SEGUNDEIRO := 0;
       #SEGUNDOS := 0;
       #MINUTEIRO := 0.0;
       #HORIMETRO := 0.0;
   END_IF;
END_REGION
END_FUNCTION_BLOCK

// ===== library: MasterCopy "FB BITS TO DOUBLE WORD" =====

// folder: 1. FB Bilbiotecas

FUNCTION_BLOCK "FB BITS TO DOUBLE WORD"   // FB5, SCL
{ S7_Optimized_Access := 'TRUE' }
VERSION : 0.1
   VAR_INPUT
      SIGNAL_Bit0 : Bool;   // Sinal de entrada 1
      SIGNAL_Bit1 : Bool;   // Sinal de entrada 2
      SIGNAL_Bit2 : Bool;   // Sinal de entrada 3
      SIGNAL_Bit3 : Bool;   // Sinal de entrada 4
      SIGNAL_Bit4 : Bool;   // Sinal de entrada 5
      SIGNAL_Bit5 : Bool;   // Sinal de entrada 6
      SIGNAL_Bit6 : Bool;   // Sinal de entrada 7
      SIGNAL_Bit7 : Bool;   // Sinal de entrada 8
      SIGNAL_Bit8 : Bool;   // Sinal de entrada 9
      SIGNAL_Bit9 : Bool;   // Sinal de entrada 10
      SIGNAL_Bit10 : Bool;   // Sinal de entrada 11
      SIGNAL_Bit11 : Bool;   // Sinal de entrada 12
      SIGNAL_Bit12 : Bool;   // Sinal de entrada 13
      SIGNAL_Bit13 : Bool;   // Sinal de entrada 14
      SIGNAL_Bit14 : Bool;   // Sinal de entrada 15
      SIGNAL_Bit15 : Bool;   // Sinal de entrada 16
      SIGNAL_Bit16 : Bool;   // Sinal de entrada 17
      SIGNAL_Bit17 : Bool;   // Sinal de entrada 18
      SIGNAL_Bit18 : Bool;   // Sinal de entrada 19
      SIGNAL_Bit19 : Bool;   // Sinal de entrada 20
      SIGNAL_Bit20 : Bool;   // Sinal de entrada 21
      SIGNAL_Bit21 : Bool;   // Sinal de entrada 22
      SIGNAL_Bit22 : Bool;   // Sinal de entrada 23
      SIGNAL_Bit23 : Bool;   // Sinal de entrada 24
      SIGNAL_Bit24 : Bool;   // Sinal de entrada 25
      SIGNAL_Bit25 : Bool;   // Sinal de entrada 26
      SIGNAL_Bit26 : Bool;   // Sinal de entrada 27
      SIGNAL_Bit27 : Bool;   // Sinal de entrada 28
      SIGNAL_Bit28 : Bool;   // Sinal de entrada 29
      SIGNAL_Bit29 : Bool;   // Sinal de entrada 30
      SIGNAL_Bit30 : Bool;   // Sinal de entrada 31
      SIGNAL_Bit31 : Bool;   // Sinal de entrada 32
   END_VAR
   VAR_OUTPUT
      BITS_TO_DWORD : DWord;   // Word de saída com os sinais montados
   END_VAR
BEGIN
   // Word Alarmes - Montando bits em uma double word

   // Bits recebidos de campo
   #"BITS_TO_DWORD".%X0 := #SIGNAL_Bit0;
   #"BITS_TO_DWORD".%X1 := #SIGNAL_Bit1;
   #"BITS_TO_DWORD".%X2 := #SIGNAL_Bit2;
   #"BITS_TO_DWORD".%X3 := #SIGNAL_Bit3;
   #"BITS_TO_DWORD".%X4 := #SIGNAL_Bit4;
   #"BITS_TO_DWORD".%X5 := #SIGNAL_Bit5;
   #"BITS_TO_DWORD".%X6 := #SIGNAL_Bit6;
   #"BITS_TO_DWORD".%X7 := #SIGNAL_Bit7;
   #"BITS_TO_DWORD".%X8 := #SIGNAL_Bit8;
   #"BITS_TO_DWORD".%X9 := #SIGNAL_Bit9;
   #"BITS_TO_DWORD".%X10 := #SIGNAL_Bit10;
   #"BITS_TO_DWORD".%X11 := #SIGNAL_Bit11;
   #"BITS_TO_DWORD".%X12 := #SIGNAL_Bit12;
   #"BITS_TO_DWORD".%X13 := #SIGNAL_Bit13;
   #"BITS_TO_DWORD".%X14 := #SIGNAL_Bit14;
   #"BITS_TO_DWORD".%X15 := #SIGNAL_Bit15;
   #"BITS_TO_DWORD".%X16 := #SIGNAL_Bit16;
   #"BITS_TO_DWORD".%X17 := #SIGNAL_Bit17;
   #"BITS_TO_DWORD".%X18 := #SIGNAL_Bit18;
   #"BITS_TO_DWORD".%X19 := #SIGNAL_Bit19;
   #"BITS_TO_DWORD".%X20 := #SIGNAL_Bit20;
   #"BITS_TO_DWORD".%X21 := #SIGNAL_Bit21;
   #"BITS_TO_DWORD".%X22 := #SIGNAL_Bit22;
   #"BITS_TO_DWORD".%X23 := #SIGNAL_Bit23;
   #"BITS_TO_DWORD".%X24 := #SIGNAL_Bit24;
   #"BITS_TO_DWORD".%X25 := #SIGNAL_Bit25;
   #"BITS_TO_DWORD".%X26 := #SIGNAL_Bit26;
   #"BITS_TO_DWORD".%X27 := #SIGNAL_Bit27;
   #"BITS_TO_DWORD".%X28 := #SIGNAL_Bit28;
   #"BITS_TO_DWORD".%X29 := #SIGNAL_Bit29;
   #"BITS_TO_DWORD".%X30 := #SIGNAL_Bit30;
   #"BITS_TO_DWORD".%X31 := #SIGNAL_Bit31;
END_FUNCTION_BLOCK

// ===== library: MasterCopy "FB_HORÍMETRO" =====

// folder: 1. FB Bilbiotecas

FUNCTION_BLOCK "FB_HORÍMETRO"   // FB22, LAD
TITLE = Function Block HORÍMETRO - Contador de Horas
{ S7_Optimized_Access := 'TRUE' }
VERSION : 0.1
// Bloco para realizar a contagem de quantas horas cada motor/bomba passou ligado.
   VAR_INPUT
      INPUT_LIGADO : Bool;   // Entrada do sinal de falha instanciado na Network 1
      INPUT_RESET_HORIMETRO : Bool;   // Entrada do sinal de reset horímetro (horas trabalhadas da bomba)
   END_VAR
   VAR_OUTPUT
      HORIMETRO : UInt;   // Saída do horímetro (horas trabalhadas da bomba)
   END_VAR
   VAR RETAIN
      RESET_SEGUNDO : Bool;   // Comando para zerar as horas acumuladas
      MINUTO : Bool;   // Pulso para contador de minutos
      COUNT_MINUTO : Bool;   // Contador de minutos
      RESET_MINUTO : Bool;   // Reset do contador de minutos
      HORA : Bool;   // Pulso para contador de horas
      COUNT_HORA : Bool;   // Contador de horas
      HORAS : UInt;   // Horas armazenadas para mover ao Horimetro e zerar quando solicitado
      TIMER_SEGUNDO : IEC_COUNTER;   // Bloco contador de segundos
      TIMER_MINUTO : IEC_COUNTER;   // Bloco contador de minutos
   END_VAR
BEGIN

REGION Network 1: Acumulação de horas (Utilizando clock de 1Hz/1s)
   // TIMER_SEGUNDO: Bloco contador de segundos
   // TIMER_MINUTO: Bloco contador de minutos
   // INC: Incremento de horas
   // RESET_HORIMETRO: Comando para zerar as horas acumuladas
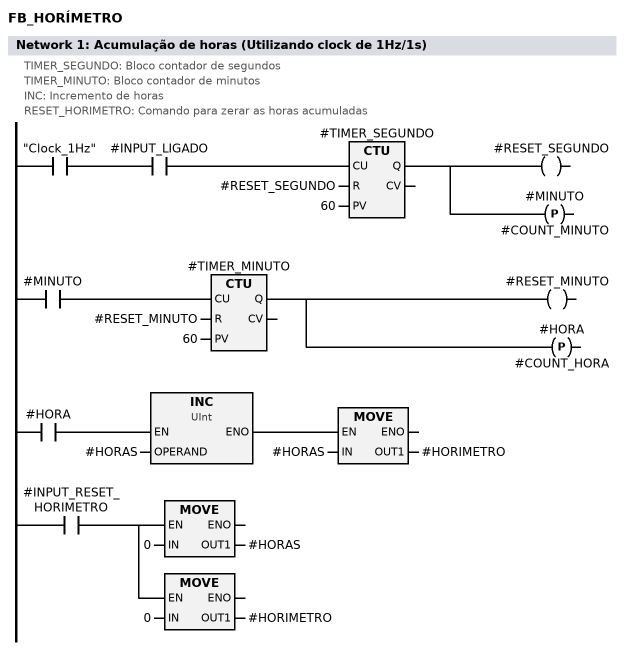
   #TIMER_SEGUNDO.CTU(CU := "Clock_1Hz" AND #INPUT_LIGADO, R := #RESET_SEGUNDO, PV := 60);
   #RESET_SEGUNDO := #TIMER_SEGUNDO.Q;
   #MINUTO := #TIMER_SEGUNDO.Q AND NOT #COUNT_MINUTO;   // rising edge
   #COUNT_MINUTO := #TIMER_SEGUNDO.Q;
   #TIMER_MINUTO.CTU(CU := #MINUTO, R := #RESET_MINUTO, PV := 60);
   #RESET_MINUTO := #TIMER_MINUTO.Q;
   #HORA := #TIMER_MINUTO.Q AND NOT #COUNT_HORA;   // rising edge
   #COUNT_HORA := #TIMER_MINUTO.Q;
   IF #HORA THEN
       #HORAS := #HORAS + 1;
       #HORIMETRO := #HORAS;
   END_IF;
   IF #INPUT_RESET_HORIMETRO THEN
       #HORAS := 0;
       #HORIMETRO := 0;
   END_IF;
END_REGION
END_FUNCTION_BLOCK

// ===== library: MasterCopy "FB TOTALIZADOR" =====

// folder: 1. FB Bilbiotecas

FUNCTION_BLOCK "FB TOTALIZADOR"   // FB16, LAD
TITLE = Function Block TOTALIZADOR - Calculando os totalizadores dos macromedidores
{ S7_Optimized_Access := 'TRUE' }
VERSION : 0.1
// Network 1: Recebendo sinal de pulso
// Network 2: Primeira Soma (Incremento a cada 1 pulso)
// Network 3: Segunda Soma (Incremento a cada 1000 pulsos)
// Network 4: Resetando o totalizador
   VAR_INPUT
      ENTRADA_SINAL : Bool;   // Entrada do sinal proveniente do hidrômetro/macromedidor
      RESET_TOT : Bool;   // Input de reset para zerar os blocos de incremento do totalizador
      MULTIPLICADOR : Int;
   END_VAR
   VAR_OUTPUT
      TOT_SAÍDA : UInt;   // Saída real do totalizador (m³)
   END_VAR
   VAR RETAIN
      PULSE1 : Bool;   // Pulso inicial para contar os sinais elétricos da entrada digital
      COUNT_PULSE1 : Bool;   // Contador de Pulsos 1
      PULSE2 : Bool;   // Rampa de subida para assegurar que o sinal da comparação anterior seja identificado como pulso pelo CLP
      COUNT_PULSE2 : Bool;   // Contador de pulsos 2
      SOMA1 : UInt;   // Bloco de incremento a cada pulso recebido na variável PULSE
      SOMA1_TOT_PREV : UInt;   // Variável que recebe a primeira soma
      SOMA2 : UInt;   // Variável que recebe o incremento de 1000 em 1000 e move ao TOT_SAÍDA Output para ser utilizado
   END_VAR
   VAR
      MULT1 : UInt;
   END_VAR
BEGIN

REGION Network 1: Recebendo sinal de pulso
   // ENTRADA_SINAL: Input que recebe o sinal de pulso do equipamento
   // PULSE1: Rampa de subida para assegurar que o sinal recebido seja identificado como pulso pelo CLP
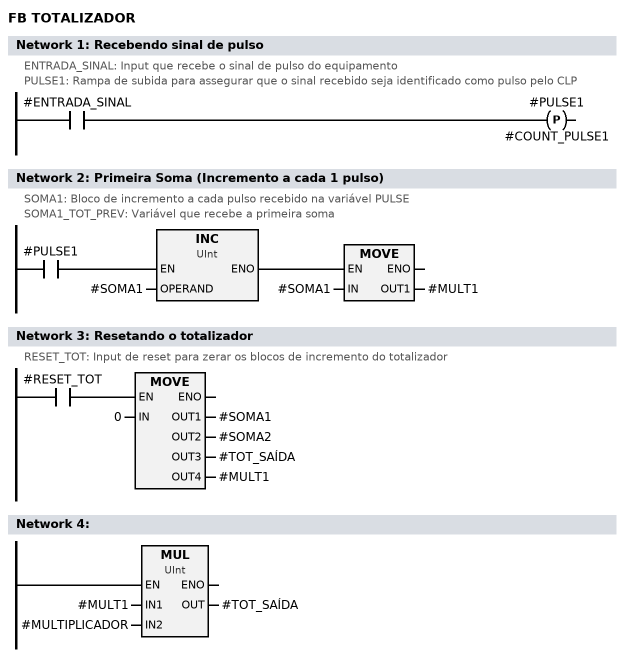
   #PULSE1 := #ENTRADA_SINAL AND NOT #COUNT_PULSE1;   // rising edge
   #COUNT_PULSE1 := #ENTRADA_SINAL;
END_REGION

REGION Network 2: Primeira Soma (Incremento a cada 1 pulso)
   // SOMA1: Bloco de incremento a cada pulso recebido na variável PULSE
   // SOMA1_TOT_PREV: Variável que recebe a primeira soma
   RUNG wire#powerrail
      Contact( #PULSE1 )
      { S7_Templates := "DestType := UInt" } Inc( #SOMA1 )
      Move(in := #SOMA1, out1 => #MULT1)
   END_RUNG
   // the same network as SCL:
   IF #PULSE1 THEN
       #SOMA1 := #SOMA1 + 1;
       #MULT1 := #SOMA1;
   END_IF;
END_REGION

